LIN {X 0,Y 360.416,Z 365.132,A -85,B 0,C 180,E1 -13245.841,E2 -13245.841} C_VEL
LIN {X 0,Y 360.571,Z 364.155,A -85,B 0,C 180,E1 -13247.25,E2 -13247.25} C_VEL
LIN {X 0,Y 360.971,Z 361.249,A -85,B 0,C 180,E1 -13249.327,E2 -13249.327} C_VEL
LIN {X 0,Y 361.318,Z 358.82,A -85,B 0,C 180,E1 -13250.493,E2 -13250.493} C_VEL
LIN {X 0,Y 361.66,Z 355.683,A -85,B 0,C 180,E1 -13251.666,E2 -13251.666} C_VEL
LIN {X 0,Y 362.259,Z 350.688,A -85,B 0,C 180,E1 -13253.131,E2 -13253.131} C_VEL
LIN {X 0,Y 362.957,Z 344.77,A -85,B 0,C 180,E1 -13254.493,E2 -13254.493} C_VEL
LIN {X 0,Y 363.512,Z 339.656,A -85,B 0,C 180,E1 -13255.477,E2 -13255.477} C_VEL
LIN {X 0,Y 364.34,Z 332.196,A -85,B 0,C 180,E1 -13256.645,E2 -13256.645} C_VEL
LIN {X 0,Y 365.036,Z 325.448,A -85,B 0,C 180,E1 -13257.519,E2 -13257.519} C_VEL
LIN {X 0,Y 365.771,Z 317.345,A -85,B 0,C 180,E1 -13258.378,E2 -13258.378} C_VEL
LIN {X 0,Y 366.188,Z 311.806,A -85,B 0,C 180,E1 -13258.881,E2 -13258.881} C_VEL
LIN {X 0,Y 364.576,Z 302,A -85,B 0,C 180,E1 -13259.701,E2 -13259.701} C_VEL
LIN {X 0,Y 362.216,Z 292.488,A -85,B 0,C 180,E1 -13260.364,E2 -13260.364} C_VEL
LIN {X 0,Y 360.856,Z 287.319,A -85,B 0,C 180,E1 -13260.684,E2 -13260.684} C_VEL
LIN {X 0,Y 360.947,Z 284.654,A -85,B 0,C 180,E1 -13263.154,E2 -13263.154} C_VEL
LIN {X 0,Y 361.044,Z 281.193,A -85,B 0,C 180,E1 -13266.457,E2 -13266.457} C_VEL
LIN {X 0,Y 360.464,Z 280.32,A -85,B 0,C 180,E1 -13267.379,E2 -13267.379} C_VEL
LIN {X 0,Y 357.716,Z 279.131,A -85,B 0,C 180,E1 -13268.886,E2 -13268.886} C_VEL
LIN {X 0,Y 355.368,Z 278.213,A -85,B 0,C 180,E1 -13270.107,E2 -13270.107} C_VEL
LIN {X 0,Y 354.387,Z 277.418,A -85,B 0,C 180,E1 -13271.047,E2 -13271.047} C_VEL
LIN {X 0,Y 354.324,Z 277.117,A -85,B 0,C 180,E1 -13271.364,E2 -13271.364} C_VEL
LIN {X 0,Y 354.508,Z 274.121,A -85,B 0,C 180,E1 -13274.468,E2 -13274.468} C_VEL
LIN {X 0,Y 354.541,Z 273.133,A -85,B 0,C 180,E1 -13275.528,E2 -13275.528} C_VEL
LIN {X 0,Y 354.741,Z 273.111,A -85,B 0,C 180,E1 -13278.834,E2 -13278.834} C_VEL
LIN {X 0,Y 354.791,Z 273.106,A -85,B 0,C 180,E1 -13282.119,E2 -13282.119} C_VEL
LIN {X 0,Y 354.793,Z 273.105,A -85,B 0,C 180,E1 -13284.942,E2 -13284.942} C_VEL
LIN {X 0,Y 354.774,Z 273.106,A -85,B 0,C 180,E1 -13288.407,E2 -13288.407} C_VEL
LIN {X 0,Y 354.828,Z 273.097,A -85,B 0,C 180,E1 -13291.62,E2 -13291.62} C_VEL
LIN {X 0,Y 354.881,Z 273.093,A -85,B 0,C 180,E1 -13294.174,E2 -13294.174} C_VEL
LIN {X 0,Y 354.81,Z 273.101,A -85,B 0,C 180,E1 -13297.895,E2 -13297.895} C_VEL
LIN {X 0,Y 354.907,Z 273.086,A -85,B 0,C 180,E1 -13301.893,E2 -13301.893} C_VEL
LIN {X 0,Y 354.929,Z 273.082,A -85,B 0,C 180,E1 -13305.983,E2 -13305.983} C_VEL
LIN {X 0,Y 354.969,Z 273.078,A -85,B 0,C 180,E1 -13309.738,E2 -13309.738} C_VEL
LIN {X 0,Y 355.087,Z 273.062,A -85,B 0,C 180,E1 -13313.182,E2 -13313.182} C_VEL
LIN {X 0,Y 355.235,Z 273.044,A -85,B 0,C 180,E1 -13317.734,E2 -13317.734} C_VEL
LIN {X 0,Y 355.386,Z 273.029,A -85,B 0,C 180,E1 -13320.002,E2 -13320.002} C_VEL
LIN {X 0,Y 355.232,Z 273.045,A -85,B 0,C 180,E1 -13322.27,E2 -13322.27} C_VEL
LIN {X 0,Y 355.129,Z 273.058,A -85,B 0,C 180,E1 -13326.821,E2 -13326.821} C_VEL
LIN {X 0,Y 355.006,Z 273.076,A -85,B 0,C 180,E1 -13329.114,E2 -13329.114} C_VEL
LIN {X 0,Y 354.916,Z 273.087,A -85,B 0,C 180,E1 -13332.583,E2 -13332.583} C_VEL
LIN {X 0,Y 354.882,Z 273.093,A -85,B 0,C 180,E1 -13336.098,E2 -13336.098} C_VEL
LIN {X 0,Y 354.895,Z 273.091,A -85,B 0,C 180,E1 -13338.474,E2 -13338.474} C_VEL
LIN {X 0,Y 354.808,Z 273.1,A -85,B 0,C 180,E1 -13342.109,E2 -13342.109} C_VEL
LIN {X 0,Y 354.82,Z 273.103,A -85,B 0,C 180,E1 -13345.835,E2 -13345.835} C_VEL
LIN {X 0,Y 354.793,Z 273.107,A -85,B 0,C 180,E1 -13349.686,E2 -13349.686} C_VEL
LIN {X 0,Y 354.781,Z 273.111,A -85,B 0,C 180,E1 -13352.336,E2 -13352.336} C_VEL
LIN {X 0,Y 354.817,Z 273.106,A -85,B 0,C 180,E1 -13355.701,E2 -13355.701} C_VEL
LIN {X 0,Y 354.82,Z 273.101,A -85,B 0,C 180,E1 -13359.426,E2 -13359.426} C_VEL
LIN {X 0,Y 354.801,Z 273.104,A -85,B 0,C 180,E1 -13362.872,E2 -13362.872} C_VEL
LIN {X 0,Y 354.763,Z 273.105,A -85,B 0,C 180,E1 -13366.106,E2 -13366.106} C_VEL
LIN {X 0,Y 354.82,Z 273.147,A -85,B 0,C 180,E1 -13367.669,E2 -13367.669} C_VEL
LIN {X 0,Y 355.607,Z 277.448,A -85,B 0,C 180,E1 -13370.773,E2 -13370.773} C_VEL
LIN {X 0,Y 356.383,Z 282.197,A -85,B 0,C 180,E1 -13373.955,E2 -13373.955} C_VEL
LIN {X 0,Y 356.829,Z 286.286,A -85,B 0,C 180,E1 -13376.534,E2 -13376.534} C_VEL
LIN {X 0,Y 356.512,Z 289.72,A -85,B 0,C 180,E1 -13378.545,E2 -13378.545} C_VEL
LIN {X 0,Y 355.735,Z 295.338,A -85,B 0,C 180,E1 -13381.698,E2 -13381.698} C_VEL
LIN {X 0,Y 354.922,Z 302.58,A -85,B 0,C 180,E1 -13385.628,E2 -13385.628} C_VEL
LIN {X 0,Y 354.219,Z 310.283,A -85,B 0,C 180,E1 -13389.685,E2 -13389.685} C_VEL
LIN {X 0,Y 353.865,Z 316.532,A -85,B 0,C 180,E1 -13392.893,E2 -13392.893} C_VEL
LIN {X 0,Y 356.246,Z 330.063,A -85,B 0,C 180,E1 -13393.674,E2 -13393.674} C_VEL
LIN {X 0,Y 357.341,Z 339.073,A -85,B 0,C 180,E1 -13394.341,E2 -13394.341} C_VEL
LIN {X 0,Y 357.782,Z 346.729,A -85,B 0,C 180,E1 -13395.013,E2 -13395.013} C_VEL
LIN {X 0,Y 357.533,Z 354.246,A -85,B 0,C 180,E1 -13395.778,E2 -13395.778} C_VEL
LIN {X 0,Y 356.617,Z 362.305,A -85,B 0,C 180,E1 -13396.758,E2 -13396.758} C_VEL
LIN {X 0,Y 355.84,Z 368.979,A -85,B 0,C 180,E1 -13397.743,E2 -13397.743} C_VEL
LIN {X 0,Y 355.12,Z 375.328,A -85,B 0,C 180,E1 -13398.876,E2 -13398.876} C_VEL
LIN {X 0,Y 354.531,Z 380.62,A -85,B 0,C 180,E1 -13400.013,E2 -13400.013} C_VEL
LIN {X 0,Y 353.96,Z 386.01,A -85,B 0,C 180,E1 -13401.438,E2 -13401.438} C_VEL
LIN {X 0,Y 353.643,Z 389.518,A -85,B 0,C 180,E1 -13402.58,E2 -13402.58} C_VEL
LIN {X 0,Y 353.349,Z 393.573,A -85,B 0,C 180,E1 -13404.294,E2 -13404.294} C_VEL
LIN {X 0,Y 353.337,Z 395.563,A -85,B 0,C 180,E1 -13405.438,E2 -13405.438} C_VEL
LIN {X 0,Y 353.267,Z 397.05,A -85,B 0,C 180,E1 -13406.58,E2 -13406.58} C_VEL
LIN {X 0,Y 353.258,Z 398.025,A -85,B 0,C 180,E1 -13407.721,E2 -13407.721} C_VEL
LIN {X 0,Y 353.357,Z 398.412,A -85,B 0,C 180,E1 -13408.862,E2 -13408.862} C_VEL
LIN {X 0,Y 353.398,Z 398.321,A -85,B 0,C 180,E1 -13410.001,E2 -13410.001} C_VEL
LIN {X 0,Y 353.396,Z 397.764,A -85,B 0,C 180,E1 -13411.141,E2 -13411.141} C_VEL
LIN {X 0,Y 353.307,Z 396.724,A -85,B 0,C 180,E1 -13412.282,E2 -13412.282} C_VEL
LIN {X 0,Y 353.343,Z 394.041,A -85,B 0,C 180,E1 -13413.993,E2 -13413.993} C_VEL
LIN {X 0,Y 353.358,Z 391.614,A -85,B 0,C 180,E1 -13415.136,E2 -13415.136} C_VEL
LIN {X 0,Y 353.53,Z 386.65,A -85,B 0,C 180,E1 -13416.852,E2 -13416.852} C_VEL
LIN {X 0,Y 353.733,Z 382.491,A -85,B 0,C 180,E1 -13417.996,E2 -13417.996} C_VEL
LIN {X 0,Y 354.012,Z 377.481,A -85,B 0,C 180,E1 -13419.14,E2 -13419.14} C_VEL
LIN {X 0,Y 354.39,Z 371.438,A -85,B 0,C 180,E1 -13420.283,E2 -13420.283} C_VEL
LIN {X 0,Y 354.914,Z 364.082,A -85,B 0,C 180,E1 -13421.423,E2 -13421.423} C_VEL
LIN {X 0,Y 355.487,Z 356.211,A -85,B 0,C 180,E1 -13422.417,E2 -13422.417} C_VEL
LIN {X 0,Y 355.957,Z 349.415,A -85,B 0,C 180,E1 -13423.125,E2 -13423.125} C_VEL
LIN {X 0,Y 355.74,Z 342.879,A -85,B 0,C 180,E1 -13423.715,E2 -13423.715} C_VEL
LIN {X 0,Y 354.992,Z 332.661,A -85,B 0,C 180,E1 -13424.45,E2 -13424.45} C_VEL
LIN {X 0,Y 354.116,Z 322.965,A -85,B 0,C 180,E1 -13424.972,E2 -13424.972} C_VEL
LIN {X 0,Y 353.55,Z 317.049,A -85,B 0,C 180,E1 -13425.236,E2 -13425.236} C_VEL
LIN {X 0,Y 353.827,Z 310.396,A -85,B 0,C 180,E1 -13428.532,E2 -13428.532} C_VEL
LIN {X 0,Y 354.261,Z 303.169,A -85,B 0,C 180,E1 -13432.145,E2 -13432.145} C_VEL
LIN {X 0,Y 354.802,Z 295.919,A -85,B 0,C 180,E1 -13435.836,E2 -13435.836} C_VEL
LIN {X 0,Y 355.492,Z 288.772,A -85,B 0,C 180,E1 -13439.554,E2 -13439.554} C_VEL
LIN {X 0,Y 356.216,Z 282.582,A -85,B 0,C 180,E1 -13442.86,E2 -13442.86} C_VEL
LIN {X 0,Y 355.899,Z 278.88,A -85,B 0,C 180,E1 -13444.938,E2 -13444.938} C_VEL
LIN {X 0,Y 354.887,Z 273.094,A -85,B 0,C 180,E1 -13448.415,E2 -13448.415} C_VEL
LIN {X 0,Y 354.804,Z 273.102,A -85,B 0,C 180,E1 -13452.337,E2 -13452.337} C_VEL
LIN {X 0,Y 354.777,Z 273.107,A -85,B 0,C 180,E1 -13456.103,E2 -13456.103} C_VEL
LIN {X 0,Y 354.797,Z 273.101,A -85,B 0,C 180,E1 -13459.179,E2 -13459.179} C_VEL
LIN {X 0,Y 354.816,Z 273.098,A -85,B 0,C 180,E1 -13462.403,E2 -13462.403} C_VEL
LIN {X 0,Y 354.822,Z 273.098,A -85,B 0,C 180,E1 -13464.94,E2 -13464.94} C_VEL
LIN {X 0,Y 354.803,Z 273.1,A -85,B 0,C 180,E1 -13468.405,E2 -13468.405} C_VEL
LIN {X 0,Y 354.861,Z 273.096,A -85,B 0,C 180,E1 -13471.618,E2 -13471.618} C_VEL
LIN {X 0,Y 354.909,Z 273.087,A -85,B 0,C 180,E1 -13474.172,E2 -13474.172} C_VEL
LIN {X 0,Y 354.827,Z 273.097,A -85,B 0,C 180,E1 -13477.892,E2 -13477.892} C_VEL
LIN {X 0,Y 354.899,Z 273.088,A -85,B 0,C 180,E1 -13481.907,E2 -13481.907} C_VEL
LIN {X 0,Y 354.952,Z 273.081,A -85,B 0,C 180,E1 -13485.98,E2 -13485.98} C_VEL
LIN {X 0,Y 354.964,Z 273.08,A -85,B 0,C 180,E1 -13489.734,E2 -13489.734} C_VEL
LIN {X 0,Y 355.119,Z 273.063,A -85,B 0,C 180,E1 -13493.179,E2 -13493.179} C_VEL
LIN {X 0,Y 355.25,Z 273.044,A -85,B 0,C 180,E1 -13497.73,E2 -13497.73} C_VEL
LIN {X 0,Y 355.381,Z 273.028,A -85,B 0,C 180,E1 -13499.998,E2 -13499.998} C_VEL
LIN {X 0,Y 355.252,Z 273.047,A -85,B 0,C 180,E1 -13502.265,E2 -13502.265} C_VEL
LIN {X 0,Y 355.143,Z 273.059,A -85,B 0,C 180,E1 -13506.817,E2 -13506.817} C_VEL
LIN {X 0,Y 355.02,Z 273.073,A -85,B 0,C 180,E1 -13509.11,E2 -13509.11} C_VEL
LIN {X 0,Y 354.925,Z 273.087,A -85,B 0,C 180,E1 -13512.578,E2 -13512.578} C_VEL
LIN {X 0,Y 354.892,Z 273.093,A -85,B 0,C 180,E1 -13516.093,E2 -13516.093} C_VEL
LIN {X 0,Y 354.905,Z 273.089,A -85,B 0,C 180,E1 -13518.469,E2 -13518.469} C_VEL
LIN {X 0,Y 354.835,Z 273.1,A -85,B 0,C 180,E1 -13522.103,E2 -13522.103} C_VEL
LIN {X 0,Y 354.898,Z 273.092,A -85,B 0,C 180,E1 -13525.825,E2 -13525.825} C_VEL
LIN {X 0,Y 354.815,Z 273.103,A -85,B 0,C 180,E1 -13529.679,E2 -13529.679} C_VEL
LIN {X 0,Y 354.803,Z 273.104,A -85,B 0,C 180,E1 -13533.699,E2 -13533.699} C_VEL
LIN {X 0,Y 354.797,Z 273.1,A -85,B 0,C 180,E1 -13536.456,E2 -13536.456} C_VEL
LIN {X 0,Y 354.818,Z 273.103,A -85,B 0,C 180,E1 -13539.421,E2 -13539.421} C_VEL
LIN {X 0,Y 354.835,Z 273.097,A -85,B 0,C 180,E1 -13542.874,E2 -13542.874} C_VEL
LIN {X 0,Y 354.858,Z 273.093,A -85,B 0,C 180,E1 -13546.116,E2 -13546.116} C_VEL
LIN {X 0,Y 354.847,Z 273.099,A -85,B 0,C 180,E1 -13549.186,E2 -13549.186} C_VEL
LIN {X 0,Y 354.799,Z 273.1,A -85,B 0,C 180,E1 -13552.399,E2 -13552.399} C_VEL
LIN {X 0,Y 354.802,Z 273.105,A -85,B 0,C 180,E1 -13554.938,E2 -13554.938} C_VEL
LIN {X 0,Y 354.781,Z 273.104,A -85,B 0,C 180,E1 -13558.402,E2 -13558.402} C_VEL
LIN {X 0,Y 354.841,Z 273.095,A -85,B 0,C 180,E1 -13561.617,E2 -13561.617} C_VEL
LIN {X 0,Y 354.886,Z 273.09,A -85,B 0,C 180,E1 -13564.17,E2 -13564.17} C_VEL
LIN {X 0,Y 354.835,Z 273.096,A -85,B 0,C 180,E1 -13567.893,E2 -13567.893} C_VEL
LIN {X 0,Y 354.771,Z 273.107,A -85,B 0,C 180,E1 -13570.318,E2 -13570.318} C_VEL
LIN {X 0,Y 354.639,Z 273.124,A -85,B 0,C 180,E1 -13572.705,E2 -13572.705} C_VEL
LIN {X 0,Y 354.215,Z 273.284,A -85,B 0,C 180,E1 -13576.447,E2 -13576.447} C_VEL
LIN {X 0,Y 354.012,Z 276.801,A -85,B 0,C 180,E1 -13579.706,E2 -13579.706} C_VEL
LIN {X 0,Y 354.09,Z 280.552,A -85,B 0,C 180,E1 -13583.159,E2 -13583.159} C_VEL
LIN {X 0,Y 353.926,Z 284.439,A -85,B 0,C 180,E1 -13586.583,E2 -13586.583} C_VEL
LIN {X 0,Y 353.759,Z 287.132,A -85,B 0,C 180,E1 -13588.931,E2 -13588.931} C_VEL
LIN {X 0,Y 355.467,Z 298.103,A -85,B 0,C 180,E1 -13589.503,E2 -13589.503} C_VEL
LIN {X 0,Y 356.869,Z 307.131,A -85,B 0,C 180,E1 -13590.14,E2 -13590.14} C_VEL
LIN {X 0,Y 356.601,Z 315.616,A -85,B 0,C 180,E1 -13590.845,E2 -13590.845} C_VEL
LIN {X 0,Y 356.062,Z 323.845,A -85,B 0,C 180,E1 -13591.695,E2 -13591.695} C_VEL
LIN {X 0,Y 355.513,Z 331.648,A -85,B 0,C 180,E1 -13592.69,E2 -13592.69} C_VEL
LIN {X 0,Y 355.093,Z 338.077,A -85,B 0,C 180,E1 -13593.687,E2 -13593.687} C_VEL
LIN {X 0,Y 354.526,Z 345.642,A -85,B 0,C 180,E1 -13595.116,E2 -13595.116} C_VEL
LIN {X 0,Y 354.214,Z 351.587,A -85,B 0,C 180,E1 -13596.549,E2 -13596.549} C_VEL
LIN {X 0,Y 353.827,Z 356.276,A -85,B 0,C 180,E1 -13597.991,E2 -13597.991} C_VEL
LIN {X 0,Y 353.593,Z 359.314,A -85,B 0,C 180,E1 -13599.148,E2 -13599.148} C_VEL
LIN {X 0,Y 353.412,Z 361.677,A -85,B 0,C 180,E1 -13600.308,E2 -13600.308} C_VEL
LIN {X 0,Y 353.348,Z 363.44,A -85,B 0,C 180,E1 -13601.471,E2 -13601.471} C_VEL
LIN {X 0,Y 353.272,Z 364.919,A -85,B 0,C 180,E1 -13602.903,E2 -13602.903} C_VEL
LIN {X 0,Y 353.249,Z 365.717,A -85,B 0,C 180,E1 -13604.988,E2 -13604.988} C_VEL
LIN {X 0,Y 353.362,Z 365.406,A -85,B 0,C 180,E1 -13606.166,E2 -13606.166} C_VEL
LIN {X 0,Y 353.516,Z 364.468,A -85,B 0,C 180,E1 -13607.408,E2 -13607.408} C_VEL
LIN {X 0,Y 353.722,Z 363.108,A -85,B 0,C 180,E1 -13608.534,E2 -13608.534} C_VEL
LIN {X 0,Y 354.198,Z 359.965,A -85,B 0,C 180,E1 -13610.316,E2 -13610.316} C_VEL
LIN {X 0,Y 354.757,Z 355.346,A -85,B 0,C 180,E1 -13612.109,E2 -13612.109} C_VEL
LIN {X 0,Y 355.445,Z 350.134,A -85,B 0,C 180,E1 -13613.601,E2 -13613.601} C_VEL
LIN {X 0,Y 356.082,Z 345.008,A -85,B 0,C 180,E1 -13614.79,E2 -13614.79} C_VEL
LIN {X 0,Y 356.705,Z 338.68,A -85,B 0,C 180,E1 -13615.999,E2 -13615.999} C_VEL
LIN {X 0,Y 357.586,Z 332.042,A -85,B 0,C 180,E1 -13617.031,E2 -13617.031} C_VEL
LIN {X 0,Y 358.34,Z 325.174,A -85,B 0,C 180,E1 -13617.922,E2 -13617.922} C_VEL
LIN {X 0,Y 359.065,Z 317.277,A -85,B 0,C 180,E1 -13618.765,E2 -13618.765} C_VEL
LIN {X 0,Y 359.325,Z 311.85,A -85,B 0,C 180,E1 -13619.271,E2 -13619.271} C_VEL
LIN {X 0,Y 357.496,Z 301.944,A -85,B 0,C 180,E1 -13620.124,E2 -13620.124} C_VEL
LIN {X 0,Y 355.149,Z 292.733,A -85,B 0,C 180,E1 -13620.784,E2 -13620.784} C_VEL
LIN {X 0,Y 353.805,Z 287.658,A -85,B 0,C 180,E1 -13621.126,E2 -13621.126} C_VEL
LIN {X 0,Y 353.887,Z 284.831,A -85,B 0,C 180,E1 -13623.782,E2 -13623.782} C_VEL
LIN {X 0,Y 354.094,Z 280.511,A -85,B 0,C 180,E1 -13627.97,E2 -13627.97} C_VEL
LIN {X 0,Y 354.324,Z 277.117,A -85,B 0,C 180,E1 -13631.364,E2 -13631.364} C_VEL
LIN {X 0,Y 353.706,Z 276.302,A -85,B 0,C 180,E1 -13632.304,E2 -13632.304} C_VEL
LIN {X 0,Y 350.908,Z 275.228,A -85,B 0,C 180,E1 -13633.84,E2 -13633.84} C_VEL
LIN {X 0,Y 348.554,Z 274.602,A -85,B 0,C 180,E1 -13635.088,E2 -13635.088} C_VEL
LIN {X 0,Y 347.597,Z 274.201,A -85,B 0,C 180,E1 -13636.053,E2 -13636.053} C_VEL
LIN {X 0,Y 347.549,Z 274.075,A -85,B 0,C 180,E1 -13636.38,E2 -13636.38} C_VEL
LIN {X 0,Y 347.699,Z 273.989,A -85,B 0,C 180,E1 -13639.702,E2 -13639.702} C_VEL
LIN {X 0,Y 347.747,Z 273.986,A -85,B 0,C 180,E1 -13642.681,E2 -13642.681} C_VEL
LIN {X 0,Y 347.729,Z 273.985,A -85,B 0,C 180,E1 -13645.957,E2 -13645.957} C_VEL
LIN {X 0,Y 347.731,Z 273.983,A -85,B 0,C 180,E1 -13649.653,E2 -13649.653} C_VEL
LIN {X 0,Y 347.813,Z 273.973,A -85,B 0,C 180,E1 -13653.609,E2 -13653.609} C_VEL
LIN {X 0,Y 347.769,Z 273.975,A -85,B 0,C 180,E1 -13656.163,E2 -13656.163} C_VEL
LIN {X 0,Y 347.795,Z 273.974,A -85,B 0,C 180,E1 -13659.911,E2 -13659.911} C_VEL
LIN {X 0,Y 347.851,Z 273.964,A -85,B 0,C 180,E1 -13662.361,E2 -13662.361} C_VEL
LIN {X 0,Y 347.883,Z 273.96,A -85,B 0,C 180,E1 -13665.973,E2 -13665.973} C_VEL
LIN {X 0,Y 347.919,Z 273.956,A -85,B 0,C 180,E1 -13669.528,E2 -13669.528} C_VEL
LIN {X 0,Y 348.055,Z 273.939,A -85,B 0,C 180,E1 -13673.044,E2 -13673.044} C_VEL
LIN {X 0,Y 348.198,Z 273.92,A -85,B 0,C 180,E1 -13677.689,E2 -13677.689} C_VEL
LIN {X 0,Y 348.334,Z 273.907,A -85,B 0,C 180,E1 -13680.002,E2 -13680.002} C_VEL
LIN {X 0,Y 348.195,Z 273.922,A -85,B 0,C 180,E1 -13682.316,E2 -13682.316} C_VEL
LIN {X 0,Y 348.097,Z 273.935,A -85,B 0,C 180,E1 -13686.96,E2 -13686.96} C_VEL
LIN {X 0,Y 347.959,Z 273.954,A -85,B 0,C 180,E1 -13689.301,E2 -13689.301} C_VEL
LIN {X 0,Y 347.884,Z 273.964,A -85,B 0,C 180,E1 -13692.842,E2 -13692.842} C_VEL
LIN {X 0,Y 347.831,Z 273.972,A -85,B 0,C 180,E1 -13696.434,E2 -13696.434} C_VEL
LIN {X 0,Y 347.844,Z 273.968,A -85,B 0,C 180,E1 -13698.863,E2 -13698.863} C_VEL
LIN {X 0,Y 347.752,Z 273.981,A -85,B 0,C 180,E1 -13702.583,E2 -13702.583} C_VEL
LIN {X 0,Y 347.769,Z 273.979,A -85,B 0,C 180,E1 -13705.114,E2 -13705.114} C_VEL
LIN {X 0,Y 347.735,Z 273.988,A -85,B 0,C 180,E1 -13707.702,E2 -13707.702} C_VEL
LIN {X 0,Y 347.735,Z 273.987,A -85,B 0,C 180,E1 -13710.351,E2 -13710.351} C_VEL
LIN {X 0,Y 347.743,Z 273.987,A -85,B 0,C 180,E1 -13714.046,E2 -13714.046} C_VEL
LIN {X 0,Y 347.758,Z 273.983,A -85,B 0,C 180,E1 -13717.323,E2 -13717.323} C_VEL
LIN {X 0,Y 347.752,Z 273.983,A -85,B 0,C 180,E1 -13720.296,E2 -13720.296} C_VEL
LIN {X 0,Y 347.741,Z 273.986,A -85,B 0,C 180,E1 -13723.407,E2 -13723.407} C_VEL
LIN {X 0,Y 347.758,Z 274.009,A -85,B 0,C 180,E1 -13727.195,E2 -13727.195} C_VEL
LIN {X 0,Y 348.479,Z 277.803,A -85,B 0,C 180,E1 -13730.031,E2 -13730.031} C_VEL
LIN {X 0,Y 349.3,Z 282.923,A -85,B 0,C 180,E1 -13733.594,E2 -13733.594} C_VEL
LIN {X 0,Y 349.785,Z 286.252,A -85,B 0,C 180,E1 -13735.767,E2 -13735.767} C_VEL
LIN {X 0,Y 349.706,Z 289.194,A -85,B 0,C 180,E1 -13737.574,E2 -13737.574} C_VEL
LIN {X 0,Y 348.863,Z 295.253,A -85,B 0,C 180,E1 -13741.088,E2 -13741.088} C_VEL
LIN {X 0,Y 347.928,Z 302.918,A -85,B 0,C 180,E1 -13745.367,E2 -13745.367} C_VEL
LIN {X 0,Y 347.212,Z 310.139,A -85,B 0,C 180,E1 -13749.256,E2 -13749.256} C_VEL
LIN {X 0,Y 346.862,Z 316.196,A -85,B 0,C 180,E1 -13752.46,E2 -13752.46} C_VEL
LIN {X 0,Y 349.142,Z 328.662,A -85,B 0,C 180,E1 -13753.182,E2 -13753.182} C_VEL
LIN {X 0,Y 350.371,Z 338.461,A -85,B 0,C 180,E1 -13753.92,E2 -13753.92} C_VEL
LIN {X 0,Y 350.919,Z 347.311,A -85,B 0,C 180,E1 -13754.727,E2 -13754.727} C_VEL
LIN {X 0,Y 350.678,Z 354.545,A -85,B 0,C 180,E1 -13755.494,E2 -13755.494} C_VEL
LIN {X 0,Y 349.733,Z 362.497,A -85,B 0,C 180,E1 -13756.492,E2 -13756.492} C_VEL
LIN {X 0,Y 348.911,Z 369.085,A -85,B 0,C 180,E1 -13757.496,E2 -13757.496} C_VEL
LIN {X 0,Y 348.147,Z 375.36,A -85,B 0,C 180,E1 -13758.65,E2 -13758.65} C_VEL
LIN {X 0,Y 347.519,Z 380.589,A -85,B 0,C 180,E1 -13759.809,E2 -13759.809} C_VEL
LIN {X 0,Y 346.918,Z 385.924,A -85,B 0,C 180,E1 -13761.262,E2 -13761.262} C_VEL
LIN {X 0,Y 346.572,Z 389.38,A -85,B 0,C 180,E1 -13762.427,E2 -13762.427} C_VEL
LIN {X 0,Y 346.273,Z 393.387,A -85,B 0,C 180,E1 -13764.177,E2 -13764.177} C_VEL
LIN {X 0,Y 346.25,Z 395.333,A -85,B 0,C 180,E1 -13765.345,E2 -13765.345} C_VEL
LIN {X 0,Y 346.19,Z 396.779,A -85,B 0,C 180,E1 -13766.51,E2 -13766.51} C_VEL
LIN {X 0,Y 346.164,Z 397.734,A -85,B 0,C 180,E1 -13767.674,E2 -13767.674} C_VEL
LIN {X 0,Y 346.258,Z 398.101,A -85,B 0,C 180,E1 -13768.839,E2 -13768.839} C_VEL
LIN {X 0,Y 346.319,Z 397.971,A -85,B 0,C 180,E1 -13770.002,E2 -13770.002} C_VEL
LIN {X 0,Y 346.3,Z 397.374,A -85,B 0,C 180,E1 -13771.164,E2 -13771.164} C_VEL
LIN {X 0,Y 346.212,Z 396.296,A -85,B 0,C 180,E1 -13772.328,E2 -13772.328} C_VEL
LIN {X 0,Y 346.274,Z 393.57,A -85,B 0,C 180,E1 -13774.075,E2 -13774.075} C_VEL
LIN {X 0,Y 346.294,Z 389.563,A -85,B 0,C 180,E1 -13775.826,E2 -13775.826} C_VEL
LIN {X 0,Y 346.456,Z 386.081,A -85,B 0,C 180,E1 -13776.992,E2 -13776.992} C_VEL
LIN {X 0,Y 346.742,Z 380.681,A -85,B 0,C 180,E1 -13778.452,E2 -13778.452} C_VEL
LIN {X 0,Y 347.145,Z 373.928,A -85,B 0,C 180,E1 -13779.91,E2 -13779.91} C_VEL
LIN {X 0,Y 347.75,Z 365.286,A -85,B 0,C 180,E1 -13781.366,E2 -13781.366} C_VEL
LIN {X 0,Y 348.312,Z 357.723,A -85,B 0,C 180,E1 -13782.381,E2 -13782.381} C_VEL
LIN {X 0,Y 348.921,Z 349.822,A -85,B 0,C 180,E1 -13783.246,E2 -13783.246} C_VEL
LIN {X 0,Y 348.599,Z 341.532,A -85,B 0,C 180,E1 -13784.002,E2 -13784.002} C_VEL
LIN {X 0,Y 348.004,Z 333.338,A -85,B 0,C 180,E1 -13784.607,E2 -13784.607} C_VEL
LIN {X 0,Y 347.135,Z 323.58,A -85,B 0,C 180,E1 -13785.159,E2 -13785.159} C_VEL
LIN {X 0,Y 346.498,Z 316.756,A -85,B 0,C 180,E1 -13785.478,E2 -13785.478} C_VEL
LIN {X 0,Y 346.753,Z 309.946,A -85,B 0,C 180,E1 -13788.924,E2 -13788.924} C_VEL
LIN {X 0,Y 347.236,Z 302.74,A -85,B 0,C 180,E1 -13792.618,E2 -13792.618} C_VEL
LIN {X 0,Y 347.827,Z 295.491,A -85,B 0,C 180,E1 -13796.394,E2 -13796.394} C_VEL
LIN {X 0,Y 348.625,Z 288.264,A -85,B 0,C 180,E1 -13800.265,E2 -13800.265} C_VEL
LIN {X 0,Y 349.192,Z 283.406,A -85,B 0,C 180,E1 -13802.918,E2 -13802.918} C_VEL
LIN {X 0,Y 348.845,Z 279.72,A -85,B 0,C 180,E1 -13805.043,E2 -13805.043} C_VEL
LIN {X 0,Y 347.845,Z 273.971,A -85,B 0,C 180,E1 -13808.57,E2 -13808.57} C_VEL
LIN {X 0,Y 347.76,Z 273.98,A -85,B 0,C 180,E1 -13811.83,E2 -13811.83} C_VEL
LIN {X 0,Y 347.715,Z 273.982,A -85,B 0,C 180,E1 -13815.027,E2 -13815.027} C_VEL
LIN {X 0,Y 347.76,Z 273.978,A -85,B 0,C 180,E1 -13818.397,E2 -13818.397} C_VEL
LIN {X 0,Y 347.782,Z 273.977,A -85,B 0,C 180,E1 -13822.011,E2 -13822.011} C_VEL
LIN {X 0,Y 347.754,Z 273.982,A -85,B 0,C 180,E1 -13825.536,E2 -13825.536} C_VEL
LIN {X 0,Y 347.774,Z 273.979,A -85,B 0,C 180,E1 -13829.653,E2 -13829.653} C_VEL
LIN {X 0,Y 347.862,Z 273.964,A -85,B 0,C 180,E1 -13832.744,E2 -13832.744} C_VEL
LIN {X 0,Y 347.795,Z 273.972,A -85,B 0,C 180,E1 -13836.161,E2 -13836.161} C_VEL
LIN {X 0,Y 347.809,Z 273.971,A -85,B 0,C 180,E1 -13839.907,E2 -13839.907} C_VEL
LIN {X 0,Y 347.841,Z 273.968,A -85,B 0,C 180,E1 -13843.567,E2 -13843.567} C_VEL
LIN {X 0,Y 347.898,Z 273.964,A -85,B 0,C 180,E1 -13847.159,E2 -13847.159} C_VEL
LIN {X 0,Y 347.943,Z 273.958,A -85,B 0,C 180,E1 -13850.699,E2 -13850.699} C_VEL
LIN {X 0,Y 348.085,Z 273.94,A -85,B 0,C 180,E1 -13853.04,E2 -13853.04} C_VEL
LIN {X 0,Y 348.212,Z 273.92,A -85,B 0,C 180,E1 -13857.685,E2 -13857.685} C_VEL
LIN {X 0,Y 348.332,Z 273.906,A -85,B 0,C 180,E1 -13859.998,E2 -13859.998} C_VEL
LIN {X 0,Y 348.214,Z 273.924,A -85,B 0,C 180,E1 -13862.311,E2 -13862.311} C_VEL
LIN {X 0,Y 348.111,Z 273.934,A -85,B 0,C 180,E1 -13866.955,E2 -13866.955} C_VEL
LIN {X 0,Y 347.972,Z 273.95,A -85,B 0,C 180,E1 -13869.296,E2 -13869.296} C_VEL
LIN {X 0,Y 347.893,Z 273.961,A -85,B 0,C 180,E1 -13872.837,E2 -13872.837} C_VEL
LIN {X 0,Y 347.841,Z 273.969,A -85,B 0,C 180,E1 -13876.429,E2 -13876.429} C_VEL
LIN {X 0,Y 347.854,Z 273.965,A -85,B 0,C 180,E1 -13878.858,E2 -13878.858} C_VEL
LIN {X 0,Y 347.774,Z 273.976,A -85,B 0,C 180,E1 -13882.577,E2 -13882.577} C_VEL
LIN {X 0,Y 347.811,Z 273.97,A -85,B 0,C 180,E1 -13885.106,E2 -13885.106} C_VEL
LIN {X 0,Y 347.807,Z 273.976,A -85,B 0,C 180,E1 -13887.691,E2 -13887.691} C_VEL
LIN {X 0,Y 347.747,Z 273.979,A -85,B 0,C 180,E1 -13890.345,E2 -13890.345} C_VEL
LIN {X 0,Y 347.745,Z 273.98,A -85,B 0,C 180,E1 -13894.041,E2 -13894.041} C_VEL
LIN {X 0,Y 347.762,Z 273.98,A -85,B 0,C 180,E1 -13897.317,E2 -13897.317} C_VEL
LIN {X 0,Y 347.788,Z 273.973,A -85,B 0,C 180,E1 -13900.286,E2 -13900.286} C_VEL
LIN {X 0,Y 347.812,Z 273.975,A -85,B 0,C 180,E1 -13903.39,E2 -13903.39} C_VEL
LIN {X 0,Y 347.809,Z 273.972,A -85,B 0,C 180,E1 -13906.667,E2 -13906.667} C_VEL
LIN {X 0,Y 347.777,Z 273.974,A -85,B 0,C 180,E1 -13910.163,E2 -13910.163} C_VEL
LIN {X 0,Y 347.778,Z 273.974,A -85,B 0,C 180,E1 -13914.122,E2 -13914.122} C_VEL
LIN {X 0,Y 347.727,Z 273.981,A -85,B 0,C 180,E1 -13918.083,E2 -13918.083} C_VEL
LIN {X 0,Y 347.794,Z 273.976,A -85,B 0,C 180,E1 -13920.988,E2 -13920.988} C_VEL
LIN {X 0,Y 347.819,Z 273.969,A -85,B 0,C 180,E1 -13923.605,E2 -13923.605} C_VEL
LIN {X 0,Y 347.784,Z 273.975,A -85,B 0,C 180,E1 -13926.16,E2 -13926.16} C_VEL
LIN {X 0,Y 347.831,Z 273.972,A -85,B 0,C 180,E1 -13928.671,E2 -13928.671} C_VEL
LIN {X 0,Y 347.649,Z 273.995,A -85,B 0,C 180,E1 -13932.346,E2 -13932.346} C_VEL
LIN {X 0,Y 347.159,Z 274.058,A -85,B 0,C 180,E1 -13936.329,E2 -13936.329} C_VEL
LIN {X 0,Y 346.963,Z 277.282,A -85,B 0,C 180,E1 -13939.495,E2 -13939.495} C_VEL
LIN {X 0,Y 347.053,Z 281.082,A -85,B 0,C 180,E1 -13943.02,E2 -13943.02} C_VEL
LIN {X 0,Y 346.871,Z 284.963,A -85,B 0,C 180,E1 -13946.514,E2 -13946.514} C_VEL
LIN {X 0,Y 346.724,Z 287.409,A -85,B 0,C 180,E1 -13948.692,E2 -13948.692} C_VEL
LIN {X 0,Y 348.385,Z 298.392,A -85,B 0,C 180,E1 -13949.276,E2 -13949.276} C_VEL
LIN {X 0,Y 349.667,Z 306.56,A -85,B 0,C 180,E1 -13949.855,E2 -13949.855} C_VEL
LIN {X 0,Y 349.862,Z 311.963,A -85,B 0,C 180,E1 -13950.286,E2 -13950.286} C_VEL
LIN {X 0,Y 349.167,Z 322.273,A -85,B 0,C 180,E1 -13951.296,E2 -13951.296} C_VEL
LIN {X 0,Y 348.636,Z 330.384,A -85,B 0,C 180,E1 -13952.309,E2 -13952.309} C_VEL
LIN {X 0,Y 348.191,Z 336.236,A -85,B 0,C 180,E1 -13953.18,E2 -13953.18} C_VEL
LIN {X 0,Y 347.744,Z 342.722,A -85,B 0,C 180,E1 -13954.345,E2 -13954.345} C_VEL
LIN {X 0,Y 347.303,Z 348.13,A -85,B 0,C 180,E1 -13955.514,E2 -13955.514} C_VEL
LIN {X 0,Y 347.172,Z 351.629,A -85,B 0,C 180,E1 -13956.391,E2 -13956.391} C_VEL
LIN {X 0,Y 346.712,Z 357.163,A -85,B 0,C 180,E1 -13958.156,E2 -13958.156} C_VEL
LIN {X 0,Y 346.391,Z 361.257,A -85,B 0,C 180,E1 -13959.929,E2 -13959.929} C_VEL
LIN {X 0,Y 346.229,Z 364.075,A -85,B 0,C 180,E1 -13961.71,E2 -13961.71} C_VEL
LIN {X 0,Y 346.182,Z 365.28,A -85,B 0,C 180,E1 -13962.989,E2 -13962.989} C_VEL
LIN {X 0,Y 346.133,Z 365.846,A -85,B 0,C 180,E1 -13964.101,E2 -13964.101} C_VEL
LIN {X 0,Y 346.174,Z 365.993,A -85,B 0,C 180,E1 -13965.301,E2 -13965.301} C_VEL
LIN {X 0,Y 346.329,Z 365.634,A -85,B 0,C 180,E1 -13966.503,E2 -13966.503} C_VEL
LIN {X 0,Y 346.498,Z 364.673,A -85,B 0,C 180,E1 -13967.711,E2 -13967.711} C_VEL
LIN {X 0,Y 346.882,Z 362.229,A -85,B 0,C 180,E1 -13969.528,E2 -13969.528} C_VEL
LIN {X 0,Y 347.25,Z 359.856,A -85,B 0,C 180,E1 -13970.742,E2 -13970.742} C_VEL
LIN {X 0,Y 347.873,Z 354.957,A -85,B 0,C 180,E1 -13972.571,E2 -13972.571} C_VEL
LIN {X 0,Y 348.469,Z 350.794,A -85,B 0,C 180,E1 -13973.787,E2 -13973.787} C_VEL
LIN {X 0,Y 349.239,Z 345.204,A -85,B 0,C 180,E1 -13975.108,E2 -13975.108} C_VEL
LIN {X 0,Y 349.803,Z 339.493,A -85,B 0,C 180,E1 -13976.23,E2 -13976.23} C_VEL
LIN {X 0,Y 350.839,Z 331.886,A -85,B 0,C 180,E1 -13977.433,E2 -13977.433} C_VEL
LIN {X 0,Y 351.603,Z 325.241,A -85,B 0,C 180,E1 -13978.302,E2 -13978.302} C_VEL
LIN {X 0,Y 352.318,Z 317.994,A -85,B 0,C 180,E1 -13979.091,E2 -13979.091} C_VEL
LIN {X 0,Y 352.574,Z 313.191,A -85,B 0,C 180,E1 -13979.559,E2 -13979.559} C_VEL
LIN {X 0,Y 350.689,Z 302.799,A -85,B 0,C 180,E1 -13980.493,E2 -13980.493} C_VEL
LIN {X 0,Y 348.32,Z 293.73,A -85,B 0,C 180,E1 -13981.177,E2 -13981.177} C_VEL
LIN {X 0,Y 346.754,Z 288.006,A -85,B 0,C 180,E1 -13981.571,E2 -13981.571} C_VEL
LIN {X 0,Y 346.854,Z 284.873,A -85,B 0,C 180,E1 -13984.563,E2 -13984.563} C_VEL
LIN {X 0,Y 347.066,Z 281.564,A -85,B 0,C 180,E1 -13987.844,E2 -13987.844} C_VEL
LIN {X 0,Y 347.345,Z 277.583,A -85,B 0,C 180,E1 -13991.888,E2 -13991.888} C_VEL
LIN {X 0,Y 347.497,Z 274.581,A -85,B 0,C 180,E1 -13995.059,E2 -13995.059} C_VEL
LIN {X 0,Y 347.549,Z 274.075,A -85,B 0,C 180,E1 -13996.38,E2 -13996.38} C_VEL
LIN {X 0,Y 347.294,Z 274.035,A -85,B 0,C 180,E1 -13997.027,E2 -13997.027} C_VEL
LIN {X 0,Y 345.416,Z 274.273,A -85,B 0,C 180,E1 -13998.298,E2 -13998.298} C_VEL
LIN {X 0,Y 341.742,Z 274.75,A -85,B 0,C 180,E1 -14000.201,E2 -14000.201} C_VEL
LIN {X 0,Y 340.745,Z 274.857,A -85,B 0,C 180,E1 -14001.19,E2 -14001.19} C_VEL
LIN {X 0,Y 340.686,Z 274.863,A -85,B 0,C 180,E1 -14001.524,E2 -14001.524} C_VEL
LIN {X 0,Y 340.7,Z 274.861,A -85,B 0,C 180,E1 -14004.722,E2 -14004.722} C_VEL
LIN {X 0,Y 340.679,Z 274.862,A -85,B 0,C 180,E1 -14008.957,E2 -14008.957} C_VEL
LIN {X 0,Y 340.786,Z 274.848,A -85,B 0,C 180,E1 -14013.021,E2 -14013.021} C_VEL
LIN {X 0,Y 340.737,Z 274.852,A -85,B 0,C 180,E1 -14015.64,E2 -14015.64} C_VEL
LIN {X 0,Y 340.723,Z 274.853,A -85,B 0,C 180,E1 -14019.475,E2 -14019.475} C_VEL
LIN {X 0,Y 340.843,Z 274.837,A -85,B 0,C 180,E1 -14021.986,E2 -14021.986} C_VEL
LIN {X 0,Y 340.855,Z 274.835,A -85,B 0,C 180,E1 -14025.707,E2 -14025.707} C_VEL
LIN {X 0,Y 340.862,Z 274.836,A -85,B 0,C 180,E1 -14029.308,E2 -14029.308} C_VEL
LIN {X 0,Y 341.003,Z 274.818,A -85,B 0,C 180,E1 -14032.899,E2 -14032.899} C_VEL
LIN {X 0,Y 341.159,Z 274.797,A -85,B 0,C 180,E1 -14037.641,E2 -14037.641} C_VEL
LIN {X 0,Y 341.285,Z 274.785,A -85,B 0,C 180,E1 -14040.002,E2 -14040.002} C_VEL
LIN {X 0,Y 341.157,Z 274.798,A -85,B 0,C 180,E1 -14042.363,E2 -14042.363} C_VEL
LIN {X 0,Y 341.066,Z 274.812,A -85,B 0,C 180,E1 -14047.104,E2 -14047.104} C_VEL
LIN {X 0,Y 340.864,Z 274.838,A -85,B 0,C 180,E1 -14050.696,E2 -14050.696} C_VEL
LIN {X 0,Y 340.855,Z 274.839,A -85,B 0,C 180,E1 -14054.327,E2 -14054.327} C_VEL
LIN {X 0,Y 340.83,Z 274.843,A -85,B 0,C 180,E1 -14058.469,E2 -14058.469} C_VEL
LIN {X 0,Y 340.711,Z 274.857,A -85,B 0,C 180,E1 -14061.844,E2 -14061.844} C_VEL
LIN {X 0,Y 340.745,Z 274.855,A -85,B 0,C 180,E1 -14064.84,E2 -14064.84} C_VEL
LIN {X 0,Y 340.679,Z 274.864,A -85,B 0,C 180,E1 -14068.327,E2 -14068.327} C_VEL
LIN {X 0,Y 340.689,Z 274.866,A -85,B 0,C 180,E1 -14071.047,E2 -14071.047} C_VEL
LIN {X 0,Y 340.713,Z 274.862,A -85,B 0,C 180,E1 -14075.281,E2 -14075.281} C_VEL
LIN {X 0,Y 340.709,Z 274.861,A -85,B 0,C 180,E1 -14078.389,E2 -14078.389} C_VEL
LIN {X 0,Y 340.728,Z 274.858,A -85,B 0,C 180,E1 -14082.054,E2 -14082.054} C_VEL
LIN {X 0,Y 340.65,Z 274.863,A -85,B 0,C 180,E1 -14086.229,E2 -14086.229} C_VEL
LIN {X 0,Y 340.761,Z 275.103,A -85,B 0,C 180,E1 -14086.901,E2 -14086.901} C_VEL
LIN {X 0,Y 341.575,Z 279.656,A -85,B 0,C 180,E1 -14090.372,E2 -14090.372} C_VEL
LIN {X 0,Y 342.49,Z 285.133,A -85,B 0,C 180,E1 -14094.211,E2 -14094.211} C_VEL
LIN {X 0,Y 342.844,Z 288.451,A -85,B 0,C 180,E1 -14096.396,E2 -14096.396} C_VEL
LIN {X 0,Y 342.298,Z 292.935,A -85,B 0,C 180,E1 -14099.119,E2 -14099.119} C_VEL
LIN {X 0,Y 341.556,Z 298.233,A -85,B 0,C 180,E1 -14102.227,E2 -14102.227} C_VEL
LIN {X 0,Y 340.81,Z 304.284,A -85,B 0,C 180,E1 -14105.644,E2 -14105.644} C_VEL
LIN {X 0,Y 340.123,Z 311.146,A -85,B 0,C 180,E1 -14109.437,E2 -14109.437} C_VEL
LIN {X 0,Y 339.818,Z 315.861,A -85,B 0,C 180,E1 -14111.994,E2 -14111.994} C_VEL
LIN {X 0,Y 342.31,Z 329.01,A -85,B 0,C 180,E1 -14112.793,E2 -14112.793} C_VEL
LIN {X 0,Y 343.572,Z 339.249,A -85,B 0,C 180,E1 -14113.601,E2 -14113.601} C_VEL
LIN {X 0,Y 344.068,Z 347.923,A -85,B 0,C 180,E1 -14114.429,E2 -14114.429} C_VEL
LIN {X 0,Y 343.816,Z 354.861,A -85,B 0,C 180,E1 -14115.198,E2 -14115.198} C_VEL
LIN {X 0,Y 342.976,Z 361.68,A -85,B 0,C 180,E1 -14116.07,E2 -14116.07} C_VEL
LIN {X 0,Y 342.188,Z 367.492,A -85,B 0,C 180,E1 -14116.945,E2 -14116.945} C_VEL
LIN {X 0,Y 341.381,Z 373.973,A -85,B 0,C 180,E1 -14118.121,E2 -14118.121} C_VEL
LIN {X 0,Y 340.694,Z 379.383,A -85,B 0,C 180,E1 -14119.302,E2 -14119.302} C_VEL
LIN {X 0,Y 340.112,Z 383.916,A -85,B 0,C 180,E1 -14120.486,E2 -14120.486} C_VEL
LIN {X 0,Y 339.697,Z 387.703,A -85,B 0,C 180,E1 -14121.675,E2 -14121.675} C_VEL
LIN {X 0,Y 339.303,Z 392.039,A -85,B 0,C 180,E1 -14123.461,E2 -14123.461} C_VEL
LIN {X 0,Y 339.148,Z 395.104,A -85,B 0,C 180,E1 -14125.247,E2 -14125.247} C_VEL
LIN {X 0,Y 339.115,Z 396.509,A -85,B 0,C 180,E1 -14126.437,E2 -14126.437} C_VEL
LIN {X 0,Y 339.074,Z 397.436,A -85,B 0,C 180,E1 -14127.626,E2 -14127.626} C_VEL
LIN {X 0,Y 339.16,Z 397.79,A -85,B 0,C 180,E1 -14128.814,E2 -14128.814} C_VEL
LIN {X 0,Y 339.227,Z 397.619,A -85,B 0,C 180,E1 -14130.002,E2 -14130.002} C_VEL
LIN {X 0,Y 339.204,Z 396.981,A -85,B 0,C 180,E1 -14131.189,E2 -14131.189} C_VEL
LIN {X 0,Y 339.119,Z 395.86,A -85,B 0,C 180,E1 -14132.377,E2 -14132.377} C_VEL
LIN {X 0,Y 339.205,Z 393.091,A -85,B 0,C 180,E1 -14134.16,E2 -14134.16} C_VEL
LIN {X 0,Y 339.213,Z 388.879,A -85,B 0,C 180,E1 -14136.008,E2 -14136.008} C_VEL
LIN {X 0,Y 339.521,Z 383.554,A -85,B 0,C 180,E1 -14137.734,E2 -14137.734} C_VEL
LIN {X 0,Y 339.848,Z 377.524,A -85,B 0,C 180,E1 -14139.224,E2 -14139.224} C_VEL
LIN {X 0,Y 340.249,Z 371.619,A -85,B 0,C 180,E1 -14140.414,E2 -14140.414} C_VEL
LIN {X 0,Y 340.76,Z 364.422,A -85,B 0,C 180,E1 -14141.602,E2 -14141.602} C_VEL
LIN {X 0,Y 341.375,Z 356.754,A -85,B 0,C 180,E1 -14142.637,E2 -14142.637} C_VEL
LIN {X 0,Y 341.894,Z 350.221,A -85,B 0,C 180,E1 -14143.372,E2 -14143.372} C_VEL
LIN {X 0,Y 341.582,Z 342.11,A -85,B 0,C 180,E1 -14144.143,E2 -14144.143} C_VEL
LIN {X 0,Y 340.918,Z 332.799,A -85,B 0,C 180,E1 -14144.85,E2 -14144.85} C_VEL
LIN {X 0,Y 340.094,Z 323.408,A -85,B 0,C 180,E1 -14145.393,E2 -14145.393} C_VEL
LIN {X 0,Y 339.422,Z 316.415,A -85,B 0,C 180,E1 -14145.732,E2 -14145.732} C_VEL
LIN {X 0,Y 339.692,Z 309.499,A -85,B 0,C 180,E1 -14149.333,E2 -14149.333} C_VEL
LIN {X 0,Y 340.226,Z 302.301,A -85,B 0,C 180,E1 -14153.11,E2 -14153.11} C_VEL
LIN {X 0,Y 340.852,Z 295.096,A -85,B 0,C 180,E1 -14156.977,E2 -14156.977} C_VEL
LIN {X 0,Y 341.694,Z 287.862,A -85,B 0,C 180,E1 -14160.946,E2 -14160.946} C_VEL
LIN {X 0,Y 342.063,Z 284.886,A -85,B 0,C 180,E1 -14162.605,E2 -14162.605} C_VEL
LIN {X 0,Y 341.909,Z 281.32,A -85,B 0,C 180,E1 -14164.692,E2 -14164.692} C_VEL
LIN {X 0,Y 340.891,Z 275.283,A -85,B 0,C 180,E1 -14168.423,E2 -14168.423} C_VEL
LIN {X 0,Y 340.774,Z 274.85,A -85,B 0,C 180,E1 -14168.764,E2 -14168.764} C_VEL
LIN {X 0,Y 340.686,Z 274.858,A -85,B 0,C 180,E1 -14172.904,E2 -14172.904} C_VEL
LIN {X 0,Y 340.686,Z 274.858,A -85,B 0,C 180,E1 -14177.095,E2 -14177.095} C_VEL
LIN {X 0,Y 340.709,Z 274.856,A -85,B 0,C 180,E1 -14180.247,E2 -14180.247} C_VEL
LIN {X 0,Y 340.72,Z 274.858,A -85,B 0,C 180,E1 -14183.559,E2 -14183.559} C_VEL
LIN {X 0,Y 340.702,Z 274.857,A -85,B 0,C 180,E1 -14186.153,E2 -14186.153} C_VEL
LIN {X 0,Y 340.785,Z 274.845,A -85,B 0,C 180,E1 -14190.332,E2 -14190.332} C_VEL
LIN {X 0,Y 340.815,Z 274.844,A -85,B 0,C 180,E1 -14193.019,E2 -14193.019} C_VEL
LIN {X 0,Y 340.765,Z 274.851,A -85,B 0,C 180,E1 -14195.637,E2 -14195.637} C_VEL
LIN {X 0,Y 340.74,Z 274.854,A -85,B 0,C 180,E1 -14199.472,E2 -14199.472} C_VEL
LIN {X 0,Y 340.802,Z 274.843,A -85,B 0,C 180,E1 -14201.979,E2 -14201.979} C_VEL
LIN {X 0,Y 340.879,Z 274.834,A -85,B 0,C 180,E1 -14205.704,E2 -14205.704} C_VEL
LIN {X 0,Y 340.856,Z 274.839,A -85,B 0,C 180,E1 -14209.304,E2 -14209.304} C_VEL
LIN {X 0,Y 341.053,Z 274.817,A -85,B 0,C 180,E1 -14212.896,E2 -14212.896} C_VEL
LIN {X 0,Y 341.174,Z 274.797,A -85,B 0,C 180,E1 -14217.637,E2 -14217.637} C_VEL
LIN {X 0,Y 341.282,Z 274.784,A -85,B 0,C 180,E1 -14219.998,E2 -14219.998} C_VEL
LIN {X 0,Y 341.176,Z 274.801,A -85,B 0,C 180,E1 -14222.359,E2 -14222.359} C_VEL
LIN {X 0,Y 341.08,Z 274.809,A -85,B 0,C 180,E1 -14227.099,E2 -14227.099} C_VEL
LIN {X 0,Y 340.875,Z 274.836,A -85,B 0,C 180,E1 -14230.691,E2 -14230.691} C_VEL
LIN {X 0,Y 340.866,Z 274.84,A -85,B 0,C 180,E1 -14234.322,E2 -14234.322} C_VEL
LIN {X 0,Y 340.839,Z 274.841,A -85,B 0,C 180,E1 -14238.464,E2 -14238.464} C_VEL
LIN {X 0,Y 340.755,Z 274.854,A -85,B 0,C 180,E1 -14241.854,E2 -14241.854} C_VEL
LIN {X 0,Y 340.771,Z 274.851,A -85,B 0,C 180,E1 -14245.661,E2 -14245.661} C_VEL
LIN {X 0,Y 340.727,Z 274.854,A -85,B 0,C 180,E1 -14248.318,E2 -14248.318} C_VEL
LIN {X 0,Y 340.695,Z 274.857,A -85,B 0,C 180,E1 -14251.042,E2 -14251.042} C_VEL
LIN {X 0,Y 340.715,Z 274.857,A -85,B 0,C 180,E1 -14255.276,E2 -14255.276} C_VEL
LIN {X 0,Y 340.714,Z 274.854,A -85,B 0,C 180,E1 -14258.385,E2 -14258.385} C_VEL
LIN {X 0,Y 340.72,Z 274.858,A -85,B 0,C 180,E1 -14261.301,E2 -14261.301} C_VEL
LIN {X 0,Y 340.774,Z 274.847,A -85,B 0,C 180,E1 -14264.519,E2 -14264.519} C_VEL
LIN {X 0,Y 340.743,Z 274.851,A -85,B 0,C 180,E1 -14267.942,E2 -14267.942} C_VEL
LIN {X 0,Y 340.725,Z 274.853,A -85,B 0,C 180,E1 -14270.25,E2 -14270.25} C_VEL
LIN {X 0,Y 340.7,Z 274.857,A -85,B 0,C 180,E1 -14273.556,E2 -14273.556} C_VEL
LIN {X 0,Y 340.681,Z 274.858,A -85,B 0,C 180,E1 -14276.151,E2 -14276.151} C_VEL
LIN {X 0,Y 340.763,Z 274.85,A -85,B 0,C 180,E1 -14280.33,E2 -14280.33} C_VEL
LIN {X 0,Y 340.792,Z 274.847,A -85,B 0,C 180,E1 -14283.017,E2 -14283.017} C_VEL
LIN {X 0,Y 340.75,Z 274.85,A -85,B 0,C 180,E1 -14285.636,E2 -14285.636} C_VEL
LIN {X 0,Y 340.722,Z 274.853,A -85,B 0,C 180,E1 -14289.471,E2 -14289.471} C_VEL
LIN {X 0,Y 340.645,Z 274.864,A -85,B 0,C 180,E1 -14291.971,E2 -14291.971} C_VEL
LIN {X 0,Y 340.143,Z 274.93,A -85,B 0,C 180,E1 -14296.18,E2 -14296.18} C_VEL
LIN {X 0,Y 340.082,Z 275.224,A -85,B 0,C 180,E1 -14296.859,E2 -14296.859} C_VEL
LIN {X 0,Y 339.884,Z 279.039,A -85,B 0,C 180,E1 -14300.477,E2 -14300.477} C_VEL
LIN {X 0,Y 339.99,Z 281.597,A -85,B 0,C 180,E1 -14302.874,E2 -14302.874} C_VEL
LIN {X 0,Y 339.817,Z 285.491,A -85,B 0,C 180,E1 -14306.441,E2 -14306.441} C_VEL
LIN {X 0,Y 339.675,Z 287.724,A -85,B 0,C 180,E1 -14308.442,E2 -14308.442} C_VEL
LIN {X 0,Y 341.319,Z 298.67,A -85,B 0,C 180,E1 -14309.04,E2 -14309.04} C_VEL
LIN {X 0,Y 342.724,Z 307.709,A -85,B 0,C 180,E1 -14309.705,E2 -14309.705} C_VEL
LIN {X 0,Y 342.93,Z 311.278,A -85,B 0,C 180,E1 -14309.998,E2 -14309.998} C_VEL
LIN {X 0,Y 342.244,Z 321.921,A -85,B 0,C 180,E1 -14311.028,E2 -14311.028} C_VEL
LIN {X 0,Y 341.671,Z 330.151,A -85,B 0,C 180,E1 -14312.061,E2 -14312.061} C_VEL
LIN {X 0,Y 341.076,Z 337.804,A -85,B 0,C 180,E1 -14313.247,E2 -14313.247} C_VEL
LIN {X 0,Y 340.596,Z 344.09,A -85,B 0,C 180,E1 -14314.436,E2 -14314.436} C_VEL
LIN {X 0,Y 340.209,Z 349.312,A -85,B 0,C 180,E1 -14315.63,E2 -14315.63} C_VEL
LIN {X 0,Y 340.046,Z 352.562,A -85,B 0,C 180,E1 -14316.486,E2 -14316.486} C_VEL
LIN {X 0,Y 339.728,Z 356.503,A -85,B 0,C 180,E1 -14317.726,E2 -14317.726} C_VEL
LIN {X 0,Y 339.355,Z 360.84,A -85,B 0,C 180,E1 -14319.535,E2 -14319.535} C_VEL
LIN {X 0,Y 339.186,Z 363.05,A -85,B 0,C 180,E1 -14320.746,E2 -14320.746} C_VEL
LIN {X 0,Y 339.119,Z 364.69,A -85,B 0,C 180,E1 -14321.959,E2 -14321.959} C_VEL
LIN {X 0,Y 339.073,Z 365.722,A -85,B 0,C 180,E1 -14323.178,E2 -14323.178} C_VEL
LIN {X 0,Y 339.064,Z 366.241,A -85,B 0,C 180,E1 -14324.401,E2 -14324.401} C_VEL
LIN {X 0,Y 339.11,Z 366.269,A -85,B 0,C 180,E1 -14325.628,E2 -14325.628} C_VEL
LIN {X 0,Y 339.27,Z 365.799,A -85,B 0,C 180,E1 -14326.857,E2 -14326.857} C_VEL
LIN {X 0,Y 339.475,Z 364.799,A -85,B 0,C 180,E1 -14328.09,E2 -14328.09} C_VEL
LIN {X 0,Y 339.924,Z 362.131,A -85,B 0,C 180,E1 -14329.945,E2 -14329.945} C_VEL
LIN {X 0,Y 340.326,Z 359.726,A -85,B 0,C 180,E1 -14331.161,E2 -14331.161} C_VEL
LIN {X 0,Y 340.752,Z 356.517,A -85,B 0,C 180,E1 -14332.429,E2 -14332.429} C_VEL
LIN {X 0,Y 341.51,Z 351.463,A -85,B 0,C 180,E1 -14333.979,E2 -14333.979} C_VEL
LIN {X 0,Y 342.44,Z 344.987,A -85,B 0,C 180,E1 -14335.528,E2 -14335.528} C_VEL
LIN {X 0,Y 343.194,Z 338.561,A -85,B 0,C 180,E1 -14336.775,E2 -14336.775} C_VEL
LIN {X 0,Y 344.103,Z 331.759,A -85,B 0,C 180,E1 -14337.851,E2 -14337.851} C_VEL
LIN {X 0,Y 345.129,Z 323.148,A -85,B 0,C 180,E1 -14338.96,E2 -14338.96} C_VEL
LIN {X 0,Y 345.838,Z 315.079,A -85,B 0,C 180,E1 -14339.797,E2 -14339.797} C_VEL
LIN {X 0,Y 344.155,Z 304.947,A -85,B 0,C 180,E1 -14340.778,E2 -14340.778} C_VEL
LIN {X 0,Y 341.33,Z 294.005,A -85,B 0,C 180,E1 -14341.633,E2 -14341.633} C_VEL
LIN {X 0,Y 339.71,Z 288.312,A -85,B 0,C 180,E1 -14342.049,E2 -14342.049} C_VEL
LIN {X 0,Y 339.836,Z 284.921,A -85,B 0,C 180,E1 -14345.382,E2 -14345.382} C_VEL
LIN {X 0,Y 340.051,Z 282.032,A -85,B 0,C 180,E1 -14348.315,E2 -14348.315} C_VEL
LIN {X 0,Y 340.326,Z 278.475,A -85,B 0,C 180,E1 -14351.98,E2 -14351.98} C_VEL
LIN {X 0,Y 340.467,Z 275.284,A -85,B 0,C 180,E1 -14355.43,E2 -14355.43} C_VEL
LIN {X 0,Y 340.538,Z 274.876,A -85,B 0,C 180,E1 -14357.078,E2 -14357.078} C_VEL
LIN {X 0,Y 340.674,Z 274.862,A -85,B 0,C 180,E1 -14360.248,E2 -14360.248} C_VEL
LIN {X 0,Y 340.686,Z 274.863,A -85,B 0,C 180,E1 -14361.524,E2 -14361.524} C_VEL
LIN {X 0,Y 340.063,Z 274.945,A -85,B 0,C 180,E1 -14362.511,E2 -14362.511} C_VEL
LIN {X 0,Y 337.18,Z 275.301,A -85,B 0,C 180,E1 -14364.115,E2 -14364.115} C_VEL
LIN {X 0,Y 334.72,Z 275.606,A -85,B 0,C 180,E1 -14365.414,E2 -14365.414} C_VEL
LIN {X 0,Y 333.686,Z 275.733,A -85,B 0,C 180,E1 -14366.42,E2 -14366.42} C_VEL
LIN {X 0,Y 333.616,Z 275.742,A -85,B 0,C 180,E1 -14366.761,E2 -14366.761} C_VEL
LIN {X 0,Y 333.676,Z 275.734,A -85,B 0,C 180,E1 -14369.714,E2 -14369.714} C_VEL
LIN {X 0,Y 333.722,Z 275.73,A -85,B 0,C 180,E1 -14372.402,E2 -14372.402} C_VEL
LIN {X 0,Y 333.709,Z 275.731,A -85,B 0,C 180,E1 -14375.092,E2 -14375.092} C_VEL
LIN {X 0,Y 333.66,Z 275.732,A -85,B 0,C 180,E1 -14379.021,E2 -14379.021} C_VEL
LIN {X 0,Y 333.779,Z 275.72,A -85,B 0,C 180,E1 -14381.591,E2 -14381.591} C_VEL
LIN {X 0,Y 333.794,Z 275.714,A -85,B 0,C 180,E1 -14385.579,E2 -14385.579} C_VEL
LIN {X 0,Y 333.824,Z 275.713,A -85,B 0,C 180,E1 -14389.08,E2 -14389.08} C_VEL
LIN {X 0,Y 333.955,Z 275.697,A -85,B 0,C 180,E1 -14392.748,E2 -14392.748} C_VEL
LIN {X 0,Y 333.795,Z 275.718,A -85,B 0,C 180,E1 -14395.171,E2 -14395.171} C_VEL
LIN {X 0,Y 334.096,Z 275.677,A -85,B 0,C 180,E1 -14397.591,E2 -14397.591} C_VEL
LIN {X 0,Y 334.235,Z 275.664,A -85,B 0,C 180,E1 -14400.002,E2 -14400.002} C_VEL
LIN {X 0,Y 334.094,Z 275.678,A -85,B 0,C 180,E1 -14402.413,E2 -14402.413} C_VEL
LIN {X 0,Y 334.016,Z 275.692,A -85,B 0,C 180,E1 -14407.255,E2 -14407.255} C_VEL
LIN {X 0,Y 333.827,Z 275.714,A -85,B 0,C 180,E1 -14410.924,E2 -14410.924} C_VEL
LIN {X 0,Y 333.8,Z 275.719,A -85,B 0,C 180,E1 -14414.637,E2 -14414.637} C_VEL
LIN {X 0,Y 333.789,Z 275.719,A -85,B 0,C 180,E1 -14418.657,E2 -14418.657} C_VEL
LIN {X 0,Y 333.647,Z 275.737,A -85,B 0,C 180,E1 -14422.283,E2 -14422.283} C_VEL
LIN {X 0,Y 333.694,Z 275.733,A -85,B 0,C 180,E1 -14425.096,E2 -14425.096} C_VEL
LIN {X 0,Y 333.649,Z 275.742,A -85,B 0,C 180,E1 -14428.98,E2 -14428.98} C_VEL
LIN {X 0,Y 333.638,Z 275.744,A -85,B 0,C 180,E1 -14432.589,E2 -14432.589} C_VEL
LIN {X 0,Y 333.672,Z 275.738,A -85,B 0,C 180,E1 -14436.141,E2 -14436.141} C_VEL
LIN {X 0,Y 333.667,Z 275.737,A -85,B 0,C 180,E1 -14439.191,E2 -14439.191} C_VEL
LIN {X 0,Y 333.663,Z 275.737,A -85,B 0,C 180,E1 -14442.509,E2 -14442.509} C_VEL
LIN {X 0,Y 333.619,Z 275.804,A -85,B 0,C 180,E1 -14446.263,E2 -14446.263} C_VEL
LIN {X 0,Y 334.409,Z 279.695,A -85,B 0,C 180,E1 -14449.348,E2 -14449.348} C_VEL
LIN {X 0,Y 335.167,Z 284.415,A -85,B 0,C 180,E1 -14452.828,E2 -14452.828} C_VEL
LIN {X 0,Y 335.727,Z 288.408,A -85,B 0,C 180,E1 -14455.585,E2 -14455.585} C_VEL
LIN {X 0,Y 335.79,Z 290.632,A -85,B 0,C 180,E1 -14457.034,E2 -14457.034} C_VEL
LIN {X 0,Y 334.931,Z 296.239,A -85,B 0,C 180,E1 -14460.457,E2 -14460.457} C_VEL
LIN {X 0,Y 334.137,Z 301.882,A -85,B 0,C 180,E1 -14463.79,E2 -14463.79} C_VEL
LIN {X 0,Y 333.33,Z 308.72,A -85,B 0,C 180,E1 -14467.698,E2 -14467.698} C_VEL
LIN {X 0,Y 332.822,Z 315.552,A -85,B 0,C 180,E1 -14471.516,E2 -14471.516} C_VEL
LIN {X 0,Y 335.028,Z 326.933,A -85,B 0,C 180,E1 -14472.198,E2 -14472.198} C_VEL
LIN {X 0,Y 336.453,Z 337.098,A -85,B 0,C 180,E1 -14472.998,E2 -14472.998} C_VEL
LIN {X 0,Y 337.12,Z 344.858,A -85,B 0,C 180,E1 -14473.725,E2 -14473.725} C_VEL
LIN {X 0,Y 337.143,Z 352.771,A -85,B 0,C 180,E1 -14474.588,E2 -14474.588} C_VEL
LIN {X 0,Y 336.281,Z 360.895,A -85,B 0,C 180,E1 -14475.632,E2 -14475.632} C_VEL
LIN {X 0,Y 335.283,Z 367.632,A -85,B 0,C 180,E1 -14476.671,E2 -14476.671} C_VEL
LIN {X 0,Y 334.428,Z 374.033,A -85,B 0,C 180,E1 -14477.871,E2 -14477.871} C_VEL
LIN {X 0,Y 333.706,Z 379.371,A -85,B 0,C 180,E1 -14479.076,E2 -14479.076} C_VEL
LIN {X 0,Y 333.108,Z 383.842,A -85,B 0,C 180,E1 -14480.284,E2 -14480.284} C_VEL
LIN {X 0,Y 332.655,Z 387.582,A -85,B 0,C 180,E1 -14481.497,E2 -14481.497} C_VEL
LIN {X 0,Y 332.249,Z 391.857,A -85,B 0,C 180,E1 -14483.321,E2 -14483.321} C_VEL
LIN {X 0,Y 332.051,Z 394.877,A -85,B 0,C 180,E1 -14485.145,E2 -14485.145} C_VEL
LIN {X 0,Y 332.04,Z 396.24,A -85,B 0,C 180,E1 -14486.361,E2 -14486.361} C_VEL
LIN {X 0,Y 331.988,Z 397.13,A -85,B 0,C 180,E1 -14487.575,E2 -14487.575} C_VEL
LIN {X 0,Y 332.062,Z 397.479,A -85,B 0,C 180,E1 -14488.789,E2 -14488.789} C_VEL
LIN {X 0,Y 332.135,Z 397.268,A -85,B 0,C 180,E1 -14490.002,E2 -14490.002} C_VEL
LIN {X 0,Y 332.108,Z 396.587,A -85,B 0,C 180,E1 -14491.214,E2 -14491.214} C_VEL
LIN {X 0,Y 332.03,Z 395.424,A -85,B 0,C 180,E1 -14492.428,E2 -14492.428} C_VEL
LIN {X 0,Y 332.135,Z 392.612,A -85,B 0,C 180,E1 -14494.249,E2 -14494.249} C_VEL
LIN {X 0,Y 332.146,Z 388.507,A -85,B 0,C 180,E1 -14496.075,E2 -14496.075} C_VEL
LIN {X 0,Y 332.455,Z 382.945,A -85,B 0,C 180,E1 -14497.899,E2 -14497.899} C_VEL
LIN {X 0,Y 332.805,Z 376.822,A -85,B 0,C 180,E1 -14499.421,E2 -14499.421} C_VEL
LIN {X 0,Y 333.24,Z 370.844,A -85,B 0,C 180,E1 -14500.636,E2 -14500.636} C_VEL
LIN {X 0,Y 333.753,Z 363.555,A -85,B 0,C 180,E1 -14501.849,E2 -14501.849} C_VEL
LIN {X 0,Y 334.448,Z 355.785,A -85,B 0,C 180,E1 -14502.903,E2 -14502.903} C_VEL
LIN {X 0,Y 334.883,Z 349.128,A -85,B 0,C 180,E1 -14503.654,E2 -14503.654} C_VEL
LIN {X 0,Y 334.435,Z 340.744,A -85,B 0,C 180,E1 -14504.452,E2 -14504.452} C_VEL
LIN {X 0,Y 333.814,Z 332.463,A -85,B 0,C 180,E1 -14505.087,E2 -14505.087} C_VEL
LIN {X 0,Y 333.014,Z 322.88,A -85,B 0,C 180,E1 -14505.65,E2 -14505.65} C_VEL
LIN {X 0,Y 332.345,Z 316.139,A -85,B 0,C 180,E1 -14505.958,E2 -14505.958} C_VEL
LIN {X 0,Y 332.673,Z 309.04,A -85,B 0,C 180,E1 -14509.757,E2 -14509.757} C_VEL
LIN {X 0,Y 333.118,Z 303.073,A -85,B 0,C 180,E1 -14512.975,E2 -14512.975} C_VEL
LIN {X 0,Y 333.787,Z 295.882,A -85,B 0,C 180,E1 -14516.918,E2 -14516.918} C_VEL
LIN {X 0,Y 334.527,Z 289.435,A -85,B 0,C 180,E1 -14520.528,E2 -14520.528} C_VEL
LIN {X 0,Y 335.032,Z 285.043,A -85,B 0,C 180,E1 -14523.054,E2 -14523.054} C_VEL
LIN {X 0,Y 334.799,Z 281.734,A -85,B 0,C 180,E1 -14525.046,E2 -14525.046} C_VEL
LIN {X 0,Y 333.724,Z 275.727,A -85,B 0,C 180,E1 -14528.89,E2 -14528.89} C_VEL
LIN {X 0,Y 333.642,Z 275.736,A -85,B 0,C 180,E1 -14532.5,E2 -14532.5} C_VEL
LIN {X 0,Y 333.607,Z 275.745,A -85,B 0,C 180,E1 -14535.955,E2 -14535.955} C_VEL
LIN {X 0,Y 333.658,Z 275.734,A -85,B 0,C 180,E1 -14539.315,E2 -14539.315} C_VEL
LIN {X 0,Y 333.675,Z 275.732,A -85,B 0,C 180,E1 -14543.168,E2 -14543.168} C_VEL
LIN {X 0,Y 333.684,Z 275.732,A -85,B 0,C 180,E1 -14545.341,E2 -14545.341} C_VEL
LIN {X 0,Y 333.713,Z 275.73,A -85,B 0,C 180,E1 -14549.71,E2 -14549.71} C_VEL
LIN {X 0,Y 333.754,Z 275.721,A -85,B 0,C 180,E1 -14552.4,E2 -14552.4} C_VEL
LIN {X 0,Y 333.736,Z 275.726,A -85,B 0,C 180,E1 -14555.09,E2 -14555.09} C_VEL
LIN {X 0,Y 333.68,Z 275.734,A -85,B 0,C 180,E1 -14559.017,E2 -14559.017} C_VEL
LIN {X 0,Y 333.75,Z 275.723,A -85,B 0,C 180,E1 -14561.585,E2 -14561.585} C_VEL
LIN {X 0,Y 333.818,Z 275.714,A -85,B 0,C 180,E1 -14565.575,E2 -14565.575} C_VEL
LIN {X 0,Y 333.826,Z 275.716,A -85,B 0,C 180,E1 -14569.076,E2 -14569.076} C_VEL
LIN {X 0,Y 334,Z 275.695,A -85,B 0,C 180,E1 -14572.745,E2 -14572.745} C_VEL
LIN {X 0,Y 333.812,Z 275.716,A -85,B 0,C 180,E1 -14575.167,E2 -14575.167} C_VEL
LIN {X 0,Y 334.111,Z 275.676,A -85,B 0,C 180,E1 -14577.587,E2 -14577.587} C_VEL
LIN {X 0,Y 334.234,Z 275.662,A -85,B 0,C 180,E1 -14579.998,E2 -14579.998} C_VEL
LIN {X 0,Y 334.113,Z 275.681,A -85,B 0,C 180,E1 -14582.409,E2 -14582.409} C_VEL
LIN {X 0,Y 334.03,Z 275.686,A -85,B 0,C 180,E1 -14587.25,E2 -14587.25} C_VEL
LIN {X 0,Y 333.838,Z 275.711,A -85,B 0,C 180,E1 -14590.919,E2 -14590.919} C_VEL
LIN {X 0,Y 333.811,Z 275.715,A -85,B 0,C 180,E1 -14594.632,E2 -14594.632} C_VEL
LIN {X 0,Y 333.798,Z 275.716,A -85,B 0,C 180,E1 -14598.652,E2 -14598.652} C_VEL
LIN {X 0,Y 333.693,Z 275.731,A -85,B 0,C 180,E1 -14602.275,E2 -14602.275} C_VEL
LIN {X 0,Y 333.734,Z 275.725,A -85,B 0,C 180,E1 -14606.243,E2 -14606.243} C_VEL
LIN {X 0,Y 333.688,Z 275.729,A -85,B 0,C 180,E1 -14608.971,E2 -14608.971} C_VEL
LIN {X 0,Y 333.64,Z 275.735,A -85,B 0,C 180,E1 -14612.584,E2 -14612.584} C_VEL
LIN {X 0,Y 333.673,Z 275.732,A -85,B 0,C 180,E1 -14616.136,E2 -14616.136} C_VEL
LIN {X 0,Y 333.679,Z 275.733,A -85,B 0,C 180,E1 -14619.184,E2 -14619.184} C_VEL
LIN {X 0,Y 333.697,Z 275.728,A -85,B 0,C 180,E1 -14622.51,E2 -14622.51} C_VEL
LIN {X 0,Y 333.721,Z 275.725,A -85,B 0,C 180,E1 -14625.974,E2 -14625.974} C_VEL
LIN {X 0,Y 333.693,Z 275.733,A -85,B 0,C 180,E1 -14629.302,E2 -14629.302} C_VEL
LIN {X 0,Y 333.656,Z 275.737,A -85,B 0,C 180,E1 -14633.165,E2 -14633.165} C_VEL
LIN {X 0,Y 333.663,Z 275.734,A -85,B 0,C 180,E1 -14635.338,E2 -14635.338} C_VEL
LIN {X 0,Y 333.691,Z 275.729,A -85,B 0,C 180,E1 -14639.708,E2 -14639.708} C_VEL
LIN {X 0,Y 333.732,Z 275.726,A -85,B 0,C 180,E1 -14642.399,E2 -14642.399} C_VEL
LIN {X 0,Y 333.719,Z 275.727,A -85,B 0,C 180,E1 -14645.089,E2 -14645.089} C_VEL
LIN {X 0,Y 333.67,Z 275.733,A -85,B 0,C 180,E1 -14649.017,E2 -14649.017} C_VEL
LIN {X 0,Y 333.597,Z 275.74,A -85,B 0,C 180,E1 -14651.577,E2 -14651.577} C_VEL
LIN {X 0,Y 333.189,Z 275.792,A -85,B 0,C 180,E1 -14655.336,E2 -14655.336} C_VEL
LIN {X 0,Y 333.039,Z 275.817,A -85,B 0,C 180,E1 -14656.576,E2 -14656.576} C_VEL
LIN {X 0,Y 332.828,Z 279.521,A -85,B 0,C 180,E1 -14660.273,E2 -14660.273} C_VEL
LIN {X 0,Y 332.93,Z 282.147,A -85,B 0,C 180,E1 -14662.788,E2 -14662.788} C_VEL
LIN {X 0,Y 332.763,Z 286.04,A -85,B 0,C 180,E1 -14666.366,E2 -14666.366} C_VEL
LIN {X 0,Y 332.601,Z 288.043,A -85,B 0,C 180,E1 -14668.182,E2 -14668.182} C_VEL
LIN {X 0,Y 334.41,Z 299.954,A -85,B 0,C 180,E1 -14668.869,E2 -14668.869} C_VEL
LIN {X 0,Y 335.776,Z 308.805,A -85,B 0,C 180,E1 -14669.549,E2 -14669.549} C_VEL
LIN {X 0,Y 335.846,Z 314.086,A -85,B 0,C 180,E1 -14669.998,E2 -14669.998} C_VEL
LIN {X 0,Y 335.107,Z 324.015,A -85,B 0,C 180,E1 -14671.05,E2 -14671.05} C_VEL
LIN {X 0,Y 334.534,Z 331.948,A -85,B 0,C 180,E1 -14672.105,E2 -14672.105} C_VEL
LIN {X 0,Y 333.958,Z 339.355,A -85,B 0,C 180,E1 -14673.316,E2 -14673.316} C_VEL
LIN {X 0,Y 333.353,Z 346.866,A -85,B 0,C 180,E1 -14674.836,E2 -14674.836} C_VEL
LIN {X 0,Y 332.979,Z 352.927,A -85,B 0,C 180,E1 -14676.417,E2 -14676.417} C_VEL
LIN {X 0,Y 332.584,Z 357.396,A -85,B 0,C 180,E1 -14677.893,E2 -14677.893} C_VEL
LIN {X 0,Y 332.361,Z 360.411,A -85,B 0,C 180,E1 -14679.124,E2 -14679.124} C_VEL
LIN {X 0,Y 332.084,Z 363.678,A -85,B 0,C 180,E1 -14680.978,E2 -14680.978} C_VEL
LIN {X 0,Y 332.016,Z 365.232,A -85,B 0,C 180,E1 -14682.219,E2 -14682.219} C_VEL
LIN {X 0,Y 331.975,Z 366.228,A -85,B 0,C 180,E1 -14683.465,E2 -14683.465} C_VEL
LIN {X 0,Y 331.992,Z 366.635,A -85,B 0,C 180,E1 -14684.714,E2 -14684.714} C_VEL
LIN {X 0,Y 332.05,Z 366.546,A -85,B 0,C 180,E1 -14685.969,E2 -14685.969} C_VEL
LIN {X 0,Y 332.371,Z 365.419,A -85,B 0,C 180,E1 -14687.923,E2 -14687.923} C_VEL
LIN {X 0,Y 332.793,Z 363.191,A -85,B 0,C 180,E1 -14689.747,E2 -14689.747} C_VEL
LIN {X 0,Y 333.365,Z 359.779,A -85,B 0,C 180,E1 -14691.511,E2 -14691.511} C_VEL
LIN {X 0,Y 333.91,Z 356.18,A -85,B 0,C 180,E1 -14692.914,E2 -14692.914} C_VEL
LIN {X 0,Y 334.726,Z 350.933,A -85,B 0,C 180,E1 -14694.497,E2 -14694.497} C_VEL
LIN {X 0,Y 335.512,Z 345.778,A -85,B 0,C 180,E1 -14695.754,E2 -14695.754} C_VEL
LIN {X 0,Y 336.317,Z 339.408,A -85,B 0,C 180,E1 -14697.031,E2 -14697.031} C_VEL
LIN {X 0,Y 337.285,Z 332.714,A -85,B 0,C 180,E1 -14698.126,E2 -14698.126} C_VEL
LIN {X 0,Y 338.202,Z 325.582,A -85,B 0,C 180,E1 -14699.09,E2 -14699.09} C_VEL
LIN {X 0,Y 338.989,Z 317.81,A -85,B 0,C 180,E1 -14699.957,E2 -14699.957} C_VEL
LIN {X 0,Y 338.748,Z 313.263,A -85,B 0,C 180,E1 -14700.444,E2 -14700.444} C_VEL
LIN {X 0,Y 336.67,Z 303.007,A -85,B 0,C 180,E1 -14701.415,E2 -14701.415} C_VEL
LIN {X 0,Y 334.061,Z 293.518,A -85,B 0,C 180,E1 -14702.171,E2 -14702.171} C_VEL
LIN {X 0,Y 332.697,Z 288.673,A -85,B 0,C 180,E1 -14702.538,E2 -14702.538} C_VEL
LIN {X 0,Y 332.883,Z 284.57,A -85,B 0,C 180,E1 -14706.657,E2 -14706.657} C_VEL
LIN {X 0,Y 333.178,Z 280.798,A -85,B 0,C 180,E1 -14710.595,E2 -14710.595} C_VEL
LIN {X 0,Y 333.392,Z 277.558,A -85,B 0,C 180,E1 -14714.076,E2 -14714.076} C_VEL
LIN {X 0,Y 333.426,Z 275.904,A -85,B 0,C 180,E1 -14715.931,E2 -14715.931} C_VEL
LIN {X 0,Y 333.584,Z 275.747,A -85,B 0,C 180,E1 -14719.325,E2 -14719.325} C_VEL
LIN {X 0,Y 333.635,Z 275.742,A -85,B 0,C 180,E1 -14722.35,E2 -14722.35} C_VEL
LIN {X 0,Y 333.655,Z 275.738,A -85,B 0,C 180,E1 -14725.343,E2 -14725.343} C_VEL
LIN {X 0,Y 333.616,Z 275.742,A -85,B 0,C 180,E1 -14726.761,E2 -14726.761} C_VEL
LIN {X 0,Y 332.993,Z 275.825,A -85,B 0,C 180,E1 -14727.769,E2 -14727.769} C_VEL
LIN {X 0,Y 330.177,Z 276.179,A -85,B 0,C 180,E1 -14729.411,E2 -14729.411} C_VEL
LIN {X 0,Y 327.763,Z 276.476,A -85,B 0,C 180,E1 -14730.74,E2 -14730.74} C_VEL
LIN {X 0,Y 326.72,Z 276.6,A -85,B 0,C 180,E1 -14731.769,E2 -14731.769} C_VEL
LIN {X 0,Y 326.632,Z 276.61,A -85,B 0,C 180,E1 -14732.117,E2 -14732.117} C_VEL
LIN {X 0,Y 326.671,Z 276.606,A -85,B 0,C 180,E1 -14734.629,E2 -14734.629} C_VEL
LIN {X 0,Y 326.605,Z 276.613,A -85,B 0,C 180,E1 -14738.545,E2 -14738.545} C_VEL
LIN {X 0,Y 326.729,Z 276.599,A -85,B 0,C 180,E1 -14741.179,E2 -14741.179} C_VEL
LIN {X 0,Y 326.749,Z 276.592,A -85,B 0,C 180,E1 -14745.435,E2 -14745.435} C_VEL
LIN {X 0,Y 326.76,Z 276.593,A -85,B 0,C 180,E1 -14748.841,E2 -14748.841} C_VEL
LIN {X 0,Y 326.909,Z 276.576,A -85,B 0,C 180,E1 -14752.591,E2 -14752.591} C_VEL
LIN {X 0,Y 326.761,Z 276.594,A -85,B 0,C 180,E1 -14755.067,E2 -14755.067} C_VEL
LIN {X 0,Y 327.037,Z 276.556,A -85,B 0,C 180,E1 -14757.539,E2 -14757.539} C_VEL
LIN {X 0,Y 327.187,Z 276.542,A -85,B 0,C 180,E1 -14760.002,E2 -14760.002} C_VEL
LIN {X 0,Y 327.035,Z 276.557,A -85,B 0,C 180,E1 -14762.466,E2 -14762.466} C_VEL
LIN {X 0,Y 326.987,Z 276.561,A -85,B 0,C 180,E1 -14766.171,E2 -14766.171} C_VEL
LIN {X 0,Y 326.905,Z 276.579,A -85,B 0,C 180,E1 -14768.657,E2 -14768.657} C_VEL
LIN {X 0,Y 326.729,Z 276.599,A -85,B 0,C 180,E1 -14772.424,E2 -14772.424} C_VEL
LIN {X 0,Y 326.746,Z 276.598,A -85,B 0,C 180,E1 -14774.96,E2 -14774.96} C_VEL
LIN {X 0,Y 326.725,Z 276.599,A -85,B 0,C 180,E1 -14778.84,E2 -14778.84} C_VEL
LIN {X 0,Y 326.593,Z 276.619,A -85,B 0,C 180,E1 -14782.791,E2 -14782.791} C_VEL
LIN {X 0,Y 326.633,Z 276.613,A -85,B 0,C 180,E1 -14785.49,E2 -14785.49} C_VEL
LIN {X 0,Y 326.611,Z 276.618,A -85,B 0,C 180,E1 -14789.666,E2 -14789.666} C_VEL
LIN {X 0,Y 326.612,Z 276.619,A -85,B 0,C 180,E1 -14792.948,E2 -14792.948} C_VEL
LIN {X 0,Y 326.608,Z 276.62,A -85,B 0,C 180,E1 -14795.522,E2 -14795.522} C_VEL
LIN {X 0,Y 326.629,Z 276.614,A -85,B 0,C 180,E1 -14799.234,E2 -14799.234} C_VEL
LIN {X 0,Y 326.596,Z 276.619,A -85,B 0,C 180,E1 -14802.979,E2 -14802.979} C_VEL
LIN {X 0,Y 326.563,Z 276.661,A -85,B 0,C 180,E1 -14805.735,E2 -14805.735} C_VEL
LIN {X 0,Y 327.268,Z 280.319,A -85,B 0,C 180,E1 -14808.733,E2 -14808.733} C_VEL
LIN {X 0,Y 328.118,Z 285.148,A -85,B 0,C 180,E1 -14812.423,E2 -14812.423} C_VEL
LIN {X 0,Y 328.728,Z 289.49,A -85,B 0,C 180,E1 -14815.492,E2 -14815.492} C_VEL
LIN {X 0,Y 328.615,Z 292.807,A -85,B 0,C 180,E1 -14817.681,E2 -14817.681} C_VEL
LIN {X 0,Y 327.889,Z 297.276,A -85,B 0,C 180,E1 -14820.465,E2 -14820.465} C_VEL
LIN {X 0,Y 326.935,Z 304.045,A -85,B 0,C 180,E1 -14824.539,E2 -14824.539} C_VEL
LIN {X 0,Y 326.101,Z 310.862,A -85,B 0,C 180,E1 -14828.51,E2 -14828.51} C_VEL
LIN {X 0,Y 325.802,Z 315.176,A -85,B 0,C 180,E1 -14830.985,E2 -14830.985} C_VEL
LIN {X 0,Y 328.266,Z 327.546,A -85,B 0,C 180,E1 -14831.785,E2 -14831.785} C_VEL
LIN {X 0,Y 329.653,Z 337.821,A -85,B 0,C 180,E1 -14832.636,E2 -14832.636} C_VEL
LIN {X 0,Y 330.295,Z 345.555,A -85,B 0,C 180,E1 -14833.399,E2 -14833.399} C_VEL
LIN {X 0,Y 330.305,Z 353.121,A -85,B 0,C 180,E1 -14834.261,E2 -14834.261} C_VEL
LIN {X 0,Y 329.438,Z 361.129,A -85,B 0,C 180,E1 -14835.327,E2 -14835.327} C_VEL
LIN {X 0,Y 328.387,Z 367.773,A -85,B 0,C 180,E1 -14836.386,E2 -14836.386} C_VEL
LIN {X 0,Y 327.48,Z 374.095,A -85,B 0,C 180,E1 -14837.609,E2 -14837.609} C_VEL
LIN {X 0,Y 326.729,Z 379.364,A -85,B 0,C 180,E1 -14838.839,E2 -14838.839} C_VEL
LIN {X 0,Y 326.113,Z 383.775,A -85,B 0,C 180,E1 -14840.074,E2 -14840.074} C_VEL
LIN {X 0,Y 325.432,Z 388.991,A -85,B 0,C 180,E1 -14841.932,E2 -14841.932} C_VEL
LIN {X 0,Y 325.187,Z 391.684,A -85,B 0,C 180,E1 -14843.175,E2 -14843.175} C_VEL
LIN {X 0,Y 325.009,Z 393.405,A -85,B 0,C 180,E1 -14844.111,E2 -14844.111} C_VEL
LIN {X 0,Y 324.966,Z 395.975,A -85,B 0,C 180,E1 -14846.282,E2 -14846.282} C_VEL
LIN {X 0,Y 324.904,Z 396.82,A -85,B 0,C 180,E1 -14847.522,E2 -14847.522} C_VEL
LIN {X 0,Y 324.964,Z 397.161,A -85,B 0,C 180,E1 -14848.762,E2 -14848.762} C_VEL
LIN {X 0,Y 325.043,Z 396.915,A -85,B 0,C 180,E1 -14850.002,E2 -14850.002} C_VEL
LIN {X 0,Y 325.012,Z 396.191,A -85,B 0,C 180,E1 -14851.241,E2 -14851.241} C_VEL
LIN {X 0,Y 324.944,Z 394.984,A -85,B 0,C 180,E1 -14852.481,E2 -14852.481} C_VEL
LIN {X 0,Y 325.041,Z 392.124,A -85,B 0,C 180,E1 -14854.342,E2 -14854.342} C_VEL
LIN {X 0,Y 325.038,Z 388.632,A -85,B 0,C 180,E1 -14855.938,E2 -14855.938} C_VEL
LIN {X 0,Y 325.351,Z 383.363,A -85,B 0,C 180,E1 -14857.761,E2 -14857.761} C_VEL
LIN {X 0,Y 325.744,Z 376.095,A -85,B 0,C 180,E1 -14859.627,E2 -14859.627} C_VEL
LIN {X 0,Y 326.244,Z 370.04,A -85,B 0,C 180,E1 -14860.866,E2 -14860.866} C_VEL
LIN {X 0,Y 326.8,Z 362.655,A -85,B 0,C 180,E1 -14862.105,E2 -14862.105} C_VEL
LIN {X 0,Y 327.401,Z 356.002,A -85,B 0,C 180,E1 -14863.028,E2 -14863.028} C_VEL
LIN {X 0,Y 327.856,Z 349.621,A -85,B 0,C 180,E1 -14863.778,E2 -14863.778} C_VEL
LIN {X 0,Y 327.412,Z 341.053,A -85,B 0,C 180,E1 -14864.626,E2 -14864.626} C_VEL
LIN {X 0,Y 326.718,Z 331.699,A -85,B 0,C 180,E1 -14865.36,E2 -14865.36} C_VEL
LIN {X 0,Y 325.924,Z 322.295,A -85,B 0,C 180,E1 -14865.919,E2 -14865.919} C_VEL
LIN {X 0,Y 325.284,Z 315.833,A -85,B 0,C 180,E1 -14866.233,E2 -14866.233} C_VEL
LIN {X 0,Y 325.633,Z 308.58,A -85,B 0,C 180,E1 -14870.203,E2 -14870.203} C_VEL
LIN {X 0,Y 326.105,Z 302.624,A -85,B 0,C 180,E1 -14873.498,E2 -14873.498} C_VEL
LIN {X 0,Y 326.688,Z 296.649,A -85,B 0,C 180,E1 -14876.859,E2 -14876.859} C_VEL
LIN {X 0,Y 327.577,Z 289.462,A -85,B 0,C 180,E1 -14880.993,E2 -14880.993} C_VEL
LIN {X 0,Y 327.988,Z 285.527,A -85,B 0,C 180,E1 -14883.311,E2 -14883.311} C_VEL
LIN {X 0,Y 327.675,Z 282.15,A -85,B 0,C 180,E1 -14885.408,E2 -14885.408} C_VEL
LIN {X 0,Y 326.684,Z 276.603,A -85,B 0,C 180,E1 -14889.134,E2 -14889.134} C_VEL
LIN {X 0,Y 326.572,Z 276.617,A -85,B 0,C 180,E1 -14893.526,E2 -14893.526} C_VEL
LIN {X 0,Y 326.586,Z 276.614,A -85,B 0,C 180,E1 -14897.028,E2 -14897.028} C_VEL
LIN {X 0,Y 326.621,Z 276.609,A -85,B 0,C 180,E1 -14900.773,E2 -14900.773} C_VEL
LIN {X 0,Y 326.622,Z 276.609,A -85,B 0,C 180,E1 -14904.48,E2 -14904.48} C_VEL
LIN {X 0,Y 326.618,Z 276.614,A -85,B 0,C 180,E1 -14907.455,E2 -14907.455} C_VEL
LIN {X 0,Y 326.671,Z 276.603,A -85,B 0,C 180,E1 -14910.34,E2 -14910.34} C_VEL
LIN {X 0,Y 326.7,Z 276.599,A -85,B 0,C 180,E1 -14914.515,E2 -14914.515} C_VEL
LIN {X 0,Y 326.628,Z 276.609,A -85,B 0,C 180,E1 -14918.542,E2 -14918.542} C_VEL
LIN {X 0,Y 326.673,Z 276.603,A -85,B 0,C 180,E1 -14922.469,E2 -14922.469} C_VEL
LIN {X 0,Y 326.768,Z 276.591,A -85,B 0,C 180,E1 -14926.313,E2 -14926.313} C_VEL
LIN {X 0,Y 326.791,Z 276.588,A -85,B 0,C 180,E1 -14930.091,E2 -14930.091} C_VEL
LIN {X 0,Y 326.989,Z 276.563,A -85,B 0,C 180,E1 -14933.829,E2 -14933.829} C_VEL
LIN {X 0,Y 327.052,Z 276.556,A -85,B 0,C 180,E1 -14937.535,E2 -14937.535} C_VEL
LIN {X 0,Y 327.186,Z 276.54,A -85,B 0,C 180,E1 -14939.998,E2 -14939.998} C_VEL
LIN {X 0,Y 327.053,Z 276.56,A -85,B 0,C 180,E1 -14942.461,E2 -14942.461} C_VEL
LIN {X 0,Y 326.977,Z 276.565,A -85,B 0,C 180,E1 -14946.635,E2 -14946.635} C_VEL
LIN {X 0,Y 326.818,Z 276.587,A -85,B 0,C 180,E1 -14949.904,E2 -14949.904} C_VEL
LIN {X 0,Y 326.762,Z 276.593,A -85,B 0,C 180,E1 -14953.683,E2 -14953.683} C_VEL
LIN {X 0,Y 326.701,Z 276.6,A -85,B 0,C 180,E1 -14957.525,E2 -14957.525} C_VEL
LIN {X 0,Y 326.665,Z 276.608,A -85,B 0,C 180,E1 -14960.132,E2 -14960.132} C_VEL
LIN {X 0,Y 326.652,Z 276.609,A -85,B 0,C 180,E1 -14964.126,E2 -14964.126} C_VEL
LIN {X 0,Y 326.682,Z 276.602,A -85,B 0,C 180,E1 -14966.855,E2 -14966.855} C_VEL
LIN {X 0,Y 326.632,Z 276.608,A -85,B 0,C 180,E1 -14970.607,E2 -14970.607} C_VEL
LIN {X 0,Y 326.603,Z 276.613,A -85,B 0,C 180,E1 -14974.016,E2 -14974.016} C_VEL
LIN {X 0,Y 326.626,Z 276.612,A -85,B 0,C 180,E1 -14977.236,E2 -14977.236} C_VEL
LIN {X 0,Y 326.63,Z 276.608,A -85,B 0,C 180,E1 -14980.199,E2 -14980.199} C_VEL
LIN {X 0,Y 326.651,Z 276.609,A -85,B 0,C 180,E1 -14983.506,E2 -14983.506} C_VEL
LIN {X 0,Y 326.642,Z 276.61,A -85,B 0,C 180,E1 -14987.011,E2 -14987.011} C_VEL
LIN {X 0,Y 326.636,Z 276.61,A -85,B 0,C 180,E1 -14990.763,E2 -14990.763} C_VEL
LIN {X 0,Y 326.602,Z 276.613,A -85,B 0,C 180,E1 -14994.477,E2 -14994.477} C_VEL
LIN {X 0,Y 326.596,Z 276.613,A -85,B 0,C 180,E1 -14997.453,E2 -14997.453} C_VEL
LIN {X 0,Y 326.649,Z 276.607,A -85,B 0,C 180,E1 -15000.338,E2 -15000.338} C_VEL
LIN {X 0,Y 326.679,Z 276.606,A -85,B 0,C 180,E1 -15004.514,E2 -15004.514} C_VEL
LIN {X 0,Y 326.634,Z 276.613,A -85,B 0,C 180,E1 -15008.543,E2 -15008.543} C_VEL
LIN {X 0,Y 326.549,Z 276.618,A -85,B 0,C 180,E1 -15011.247,E2 -15011.247} C_VEL
LIN {X 0,Y 326.169,Z 276.666,A -85,B 0,C 180,E1 -15015.014,E2 -15015.014} C_VEL
LIN {X 0,Y 326.031,Z 276.688,A -85,B 0,C 180,E1 -15016.282,E2 -15016.282} C_VEL
LIN {X 0,Y 325.9,Z 277.464,A -85,B 0,C 180,E1 -15017.545,E2 -15017.545} C_VEL
LIN {X 0,Y 325.762,Z 281.313,A -85,B 0,C 180,E1 -15021.313,E2 -15021.313} C_VEL
LIN {X 0,Y 325.756,Z 283.927,A -85,B 0,C 180,E1 -15023.806,E2 -15023.806} C_VEL
LIN {X 0,Y 325.71,Z 286.562,A -85,B 0,C 180,E1 -15026.287,E2 -15026.287} C_VEL
LIN {X 0,Y 325.537,Z 288.315,A -85,B 0,C 180,E1 -15027.911,E2 -15027.911} C_VEL
LIN {X 0,Y 327.392,Z 300.119,A -85,B 0,C 180,E1 -15028.615,E2 -15028.615} C_VEL
LIN {X 0,Y 328.815,Z 309.89,A -85,B 0,C 180,E1 -15029.386,E2 -15029.386} C_VEL
LIN {X 0,Y 328.838,Z 315.038,A -85,B 0,C 180,E1 -15029.845,E2 -15029.845} C_VEL
LIN {X 0,Y 328.201,Z 323.61,A -85,B 0,C 180,E1 -15030.765,E2 -15030.765} C_VEL
LIN {X 0,Y 327.571,Z 331.674,A -85,B 0,C 180,E1 -15031.843,E2 -15031.843} C_VEL
LIN {X 0,Y 327.108,Z 337.471,A -85,B 0,C 180,E1 -15032.769,E2 -15032.769} C_VEL
LIN {X 0,Y 326.598,Z 343.921,A -85,B 0,C 180,E1 -15034.009,E2 -15034.009} C_VEL
LIN {X 0,Y 326.11,Z 349.295,A -85,B 0,C 180,E1 -15035.254,E2 -15035.254} C_VEL
LIN {X 0,Y 325.976,Z 352.774,A -85,B 0,C 180,E1 -15036.187,E2 -15036.187} C_VEL
LIN {X 0,Y 325.601,Z 356.664,A -85,B 0,C 180,E1 -15037.439,E2 -15037.439} C_VEL
LIN {X 0,Y 325.218,Z 361.163,A -85,B 0,C 180,E1 -15039.326,E2 -15039.326} C_VEL
LIN {X 0,Y 324.964,Z 364.303,A -85,B 0,C 180,E1 -15041.222,E2 -15041.222} C_VEL
LIN {X 0,Y 324.897,Z 366.343,A -85,B 0,C 180,E1 -15043.256,E2 -15043.256} C_VEL
LIN {X 0,Y 324.92,Z 367.03,A -85,B 0,C 180,E1 -15045.042,E2 -15045.042} C_VEL
LIN {X 0,Y 325.008,Z 366.824,A -85,B 0,C 180,E1 -15046.325,E2 -15046.325} C_VEL
LIN {X 0,Y 325.313,Z 365.748,A -85,B 0,C 180,E1 -15048.101,E2 -15048.101} C_VEL
LIN {X 0,Y 325.847,Z 363.138,A -85,B 0,C 180,E1 -15050.186,E2 -15050.186} C_VEL
LIN {X 0,Y 326.292,Z 360.756,A -85,B 0,C 180,E1 -15051.477,E2 -15051.477} C_VEL
LIN {X 0,Y 327.072,Z 355.811,A -85,B 0,C 180,E1 -15053.421,E2 -15053.421} C_VEL
LIN {X 0,Y 327.774,Z 351.617,A -85,B 0,C 180,E1 -15054.713,E2 -15054.713} C_VEL
LIN {X 0,Y 328.655,Z 346.092,A -85,B 0,C 180,E1 -15056.094,E2 -15056.094} C_VEL
LIN {X 0,Y 329.463,Z 340.258,A -85,B 0,C 180,E1 -15057.297,E2 -15057.297} C_VEL
LIN {X 0,Y 330.579,Z 332.599,A -85,B 0,C 180,E1 -15058.575,E2 -15058.575} C_VEL
LIN {X 0,Y 331.522,Z 325.687,A -85,B 0,C 180,E1 -15059.518,E2 -15059.518} C_VEL
LIN {X 0,Y 332.3,Z 318.33,A -85,B 0,C 180,E1 -15060.355,E2 -15060.355} C_VEL
LIN {X 0,Y 331.681,Z 312.635,A -85,B 0,C 180,E1 -15060.987,E2 -15060.987} C_VEL
LIN {X 0,Y 329.844,Z 303.819,A -85,B 0,C 180,E1 -15061.852,E2 -15061.852} C_VEL
LIN {X 0,Y 327.119,Z 294.044,A -85,B 0,C 180,E1 -15062.662,E2 -15062.662} C_VEL
LIN {X 0,Y 325.647,Z 289.006,A -85,B 0,C 180,E1 -15063.043,E2 -15063.043} C_VEL
LIN {X 0,Y 325.858,Z 285.013,A -85,B 0,C 180,E1 -15067.147,E2 -15067.147} C_VEL
LIN {X 0,Y 326.171,Z 281.354,A -85,B 0,C 180,E1 -15071.054,E2 -15071.054} C_VEL
LIN {X 0,Y 326.336,Z 279.061,A -85,B 0,C 180,E1 -15073.561,E2 -15073.561} C_VEL
LIN {X 0,Y 326.369,Z 276.641,A -85,B 0,C 180,E1 -15076.447,E2 -15076.447} C_VEL
LIN {X 0,Y 326.544,Z 276.624,A -85,B 0,C 180,E1 -15079.788,E2 -15079.788} C_VEL
LIN {X 0,Y 326.613,Z 276.617,A -85,B 0,C 180,E1 -15082.955,E2 -15082.955} C_VEL
LIN {X 0,Y 326.584,Z 276.617,A -85,B 0,C 180,E1 -15086.768,E2 -15086.768} C_VEL
LIN {X 0,Y 326.63,Z 276.613,A -85,B 0,C 180,E1 -15090.341,E2 -15090.341} C_VEL
LIN {X 0,Y 326.632,Z 276.61,A -85,B 0,C 180,E1 -15092.117,E2 -15092.117} C_VEL
LIN {X 0,Y 325.964,Z 276.694,A -85,B 0,C 180,E1 -15093.146,E2 -15093.146} C_VEL
LIN {X 0,Y 323.126,Z 277.048,A -85,B 0,C 180,E1 -15094.821,E2 -15094.821} C_VEL
LIN {X 0,Y 320.712,Z 277.35,A -85,B 0,C 180,E1 -15096.177,E2 -15096.177} C_VEL
LIN {X 0,Y 319.659,Z 277.481,A -85,B 0,C 180,E1 -15097.227,E2 -15097.227} C_VEL
LIN {X 0,Y 319.564,Z 277.492,A -85,B 0,C 180,E1 -15097.583,E2 -15097.583} C_VEL
LIN {X 0,Y 319.673,Z 277.478,A -85,B 0,C 180,E1 -15100.964,E2 -15100.964} C_VEL
LIN {X 0,Y 319.716,Z 277.469,A -85,B 0,C 180,E1 -15105.278,E2 -15105.278} C_VEL
LIN {X 0,Y 319.74,Z 277.465,A -85,B 0,C 180,E1 -15109.875,E2 -15109.875} C_VEL
LIN {X 0,Y 319.896,Z 277.444,A -85,B 0,C 180,E1 -15113.696,E2 -15113.696} C_VEL
LIN {X 0,Y 319.981,Z 277.435,A -85,B 0,C 180,E1 -15117.485,E2 -15117.485} C_VEL
LIN {X 0,Y 320.139,Z 277.42,A -85,B 0,C 180,E1 -15120.002,E2 -15120.002} C_VEL
LIN {X 0,Y 319.979,Z 277.436,A -85,B 0,C 180,E1 -15122.52,E2 -15122.52} C_VEL
LIN {X 0,Y 319.942,Z 277.438,A -85,B 0,C 180,E1 -15126.308,E2 -15126.308} C_VEL
LIN {X 0,Y 319.834,Z 277.458,A -85,B 0,C 180,E1 -15128.85,E2 -15128.85} C_VEL
LIN {X 0,Y 319.675,Z 277.477,A -85,B 0,C 180,E1 -15132.702,E2 -15132.702} C_VEL
LIN {X 0,Y 319.691,Z 277.477,A -85,B 0,C 180,E1 -15135.298,E2 -15135.298} C_VEL
LIN {X 0,Y 319.666,Z 277.479,A -85,B 0,C 180,E1 -15139.258,E2 -15139.258} C_VEL
LIN {X 0,Y 319.549,Z 277.495,A -85,B 0,C 180,E1 -15143.323,E2 -15143.323} C_VEL
LIN {X 0,Y 319.567,Z 277.497,A -85,B 0,C 180,E1 -15146.096,E2 -15146.096} C_VEL
LIN {X 0,Y 319.538,Z 277.5,A -85,B 0,C 180,E1 -15148.941,E2 -15148.941} C_VEL
LIN {X 0,Y 319.519,Z 277.503,A -85,B 0,C 180,E1 -15151.865,E2 -15151.865} C_VEL
LIN {X 0,Y 319.575,Z 277.496,A -85,B 0,C 180,E1 -15155.545,E2 -15155.545} C_VEL
LIN {X 0,Y 319.577,Z 277.492,A -85,B 0,C 180,E1 -15158.009,E2 -15158.009} C_VEL
LIN {X 0,Y 319.566,Z 277.493,A -85,B 0,C 180,E1 -15161.608,E2 -15161.608} C_VEL
LIN {X 0,Y 319.513,Z 277.613,A -85,B 0,C 180,E1 -15165.264,E2 -15165.264} C_VEL
LIN {X 0,Y 320.334,Z 281.843,A -85,B 0,C 180,E1 -15168.841,E2 -15168.841} C_VEL
LIN {X 0,Y 321.086,Z 286.16,A -85,B 0,C 180,E1 -15172.205,E2 -15172.205} C_VEL
LIN {X 0,Y 321.721,Z 290.557,A -85,B 0,C 180,E1 -15175.394,E2 -15175.394} C_VEL
LIN {X 0,Y 321.593,Z 293.884,A -85,B 0,C 180,E1 -15177.63,E2 -15177.63} C_VEL
LIN {X 0,Y 320.629,Z 299.583,A -85,B 0,C 180,E1 -15181.258,E2 -15181.258} C_VEL
LIN {X 0,Y 319.669,Z 306.208,A -85,B 0,C 180,E1 -15185.311,E2 -15185.311} C_VEL
LIN {X 0,Y 318.891,Z 312.999,A -85,B 0,C 180,E1 -15189.354,E2 -15189.354} C_VEL
LIN {X 0,Y 318.791,Z 315.103,A -85,B 0,C 180,E1 -15190.466,E2 -15190.466} C_VEL
LIN {X 0,Y 321.378,Z 327.463,A -85,B 0,C 180,E1 -15191.296,E2 -15191.296} C_VEL
LIN {X 0,Y 322.691,Z 336.744,A -85,B 0,C 180,E1 -15192.081,E2 -15192.081} C_VEL
LIN {X 0,Y 323.441,Z 345.388,A -85,B 0,C 180,E1 -15192.957,E2 -15192.957} C_VEL
LIN {X 0,Y 323.504,Z 353.499,A -85,B 0,C 180,E1 -15193.921,E2 -15193.921} C_VEL
LIN {X 0,Y 322.606,Z 361.38,A -85,B 0,C 180,E1 -15195.009,E2 -15195.009} C_VEL
LIN {X 0,Y 321.504,Z 367.925,A -85,B 0,C 180,E1 -15196.088,E2 -15196.088} C_VEL
LIN {X 0,Y 320.54,Z 374.161,A -85,B 0,C 180,E1 -15197.337,E2 -15197.337} C_VEL
LIN {X 0,Y 319.764,Z 379.358,A -85,B 0,C 180,E1 -15198.593,E2 -15198.593} C_VEL
LIN {X 0,Y 319.104,Z 383.708,A -85,B 0,C 180,E1 -15199.854,E2 -15199.854} C_VEL
LIN {X 0,Y 318.393,Z 388.87,A -85,B 0,C 180,E1 -15201.753,E2 -15201.753} C_VEL
LIN {X 0,Y 317.985,Z 392.678,A -85,B 0,C 180,E1 -15203.657,E2 -15203.657} C_VEL
LIN {X 0,Y 317.871,Z 394.437,A -85,B 0,C 180,E1 -15204.928,E2 -15204.928} C_VEL
LIN {X 0,Y 317.872,Z 395.71,A -85,B 0,C 180,E1 -15206.199,E2 -15206.199} C_VEL
LIN {X 0,Y 317.823,Z 396.511,A -85,B 0,C 180,E1 -15207.467,E2 -15207.467} C_VEL
LIN {X 0,Y 317.868,Z 396.834,A -85,B 0,C 180,E1 -15208.735,E2 -15208.735} C_VEL
LIN {X 0,Y 317.951,Z 396.562,A -85,B 0,C 180,E1 -15210.002,E2 -15210.002} C_VEL
LIN {X 0,Y 317.917,Z 395.793,A -85,B 0,C 180,E1 -15211.268,E2 -15211.268} C_VEL
LIN {X 0,Y 317.862,Z 394.541,A -85,B 0,C 180,E1 -15212.536,E2 -15212.536} C_VEL
LIN {X 0,Y 317.95,Z 391.632,A -85,B 0,C 180,E1 -15214.439,E2 -15214.439} C_VEL
LIN {X 0,Y 317.954,Z 388.485,A -85,B 0,C 180,E1 -15215.906,E2 -15215.906} C_VEL
LIN {X 0,Y 318.286,Z 382.758,A -85,B 0,C 180,E1 -15217.934,E2 -15217.934} C_VEL
LIN {X 0,Y 318.642,Z 376.799,A -85,B 0,C 180,E1 -15219.523,E2 -15219.523} C_VEL
LIN {X 0,Y 319.245,Z 369.23,A -85,B 0,C 180,E1 -15221.108,E2 -15221.108} C_VEL
LIN {X 0,Y 319.746,Z 362.78,A -85,B 0,C 180,E1 -15222.215,E2 -15222.215} C_VEL
LIN {X 0,Y 320.354,Z 356.218,A -85,B 0,C 180,E1 -15223.158,E2 -15223.158} C_VEL
LIN {X 0,Y 320.834,Z 349.767,A -85,B 0,C 180,E1 -15223.945,E2 -15223.945} C_VEL
LIN {X 0,Y 320.39,Z 341.564,A -85,B 0,C 180,E1 -15224.79,E2 -15224.79} C_VEL
LIN {X 0,Y 319.744,Z 332.447,A -85,B 0,C 180,E1 -15225.54,E2 -15225.54} C_VEL
LIN {X 0,Y 318.897,Z 322.579,A -85,B 0,C 180,E1 -15226.156,E2 -15226.156} C_VEL
LIN {X 0,Y 318.189,Z 315.49,A -85,B 0,C 180,E1 -15226.523,E2 -15226.523} C_VEL
LIN {X 0,Y 318.522,Z 309.311,A -85,B 0,C 180,E1 -15230,E2 -15230} C_VEL
LIN {X 0,Y 319.022,Z 303.351,A -85,B 0,C 180,E1 -15233.363,E2 -15233.363} C_VEL
LIN {X 0,Y 319.605,Z 297.417,A -85,B 0,C 180,E1 -15236.796,E2 -15236.796} C_VEL
LIN {X 0,Y 320.352,Z 291.428,A -85,B 0,C 180,E1 -15240.305,E2 -15240.305} C_VEL
LIN {X 0,Y 320.928,Z 286.631,A -85,B 0,C 180,E1 -15243.196,E2 -15243.196} C_VEL
LIN {X 0,Y 320.556,Z 282.563,A -85,B 0,C 180,E1 -15245.784,E2 -15245.784} C_VEL
LIN {X 0,Y 319.648,Z 277.48,A -85,B 0,C 180,E1 -15249.208,E2 -15249.208} C_VEL
LIN {X 0,Y 319.532,Z 277.494,A -85,B 0,C 180,E1 -15253.46,E2 -15253.46} C_VEL
LIN {X 0,Y 319.564,Z 277.488,A -85,B 0,C 180,E1 -15257.016,E2 -15257.016} C_VEL
LIN {X 0,Y 319.557,Z 277.49,A -85,B 0,C 180,E1 -15260.37,E2 -15260.37} C_VEL
LIN {X 0,Y 319.568,Z 277.492,A -85,B 0,C 180,E1 -15263.572,E2 -15263.572} C_VEL
LIN {X 0,Y 319.588,Z 277.485,A -85,B 0,C 180,E1 -15266.686,E2 -15266.686} C_VEL
LIN {X 0,Y 319.602,Z 277.488,A -85,B 0,C 180,E1 -15269.616,E2 -15269.616} C_VEL
LIN {X 0,Y 319.619,Z 277.481,A -85,B 0,C 180,E1 -15272.497,E2 -15272.497} C_VEL
LIN {X 0,Y 319.614,Z 277.487,A -85,B 0,C 180,E1 -15275.303,E2 -15275.303} C_VEL
LIN {X 0,Y 319.592,Z 277.489,A -85,B 0,C 180,E1 -15279.398,E2 -15279.398} C_VEL
LIN {X 0,Y 319.66,Z 277.479,A -85,B 0,C 180,E1 -15283.39,E2 -15283.39} C_VEL
LIN {X 0,Y 319.741,Z 277.466,A -85,B 0,C 180,E1 -15286.006,E2 -15286.006} C_VEL
LIN {X 0,Y 319.744,Z 277.466,A -85,B 0,C 180,E1 -15289.87,E2 -15289.87} C_VEL
LIN {X 0,Y 319.943,Z 277.441,A -85,B 0,C 180,E1 -15293.692,E2 -15293.692} C_VEL
LIN {X 0,Y 319.996,Z 277.434,A -85,B 0,C 180,E1 -15297.48,E2 -15297.48} C_VEL
LIN {X 0,Y 320.138,Z 277.417,A -85,B 0,C 180,E1 -15299.998,E2 -15299.998} C_VEL
LIN {X 0,Y 319.997,Z 277.44,A -85,B 0,C 180,E1 -15302.515,E2 -15302.515} C_VEL
LIN {X 0,Y 319.937,Z 277.443,A -85,B 0,C 180,E1 -15306.625,E2 -15306.625} C_VEL
LIN {X 0,Y 319.762,Z 277.467,A -85,B 0,C 180,E1 -15310.124,E2 -15310.124} C_VEL
LIN {X 0,Y 319.734,Z 277.468,A -85,B 0,C 180,E1 -15314.721,E2 -15314.721} C_VEL
LIN {X 0,Y 319.691,Z 277.472,A -85,B 0,C 180,E1 -15319.035,E2 -15319.035} C_VEL
LIN {X 0,Y 319.571,Z 277.488,A -85,B 0,C 180,E1 -15323.316,E2 -15323.316} C_VEL
LIN {X 0,Y 319.633,Z 277.483,A -85,B 0,C 180,E1 -15326.085,E2 -15326.085} C_VEL
LIN {X 0,Y 319.578,Z 277.487,A -85,B 0,C 180,E1 -15328.931,E2 -15328.931} C_VEL
LIN {X 0,Y 319.528,Z 277.497,A -85,B 0,C 180,E1 -15331.859,E2 -15331.859} C_VEL
LIN {X 0,Y 319.577,Z 277.492,A -85,B 0,C 180,E1 -15335.54,E2 -15335.54} C_VEL
LIN {X 0,Y 319.596,Z 277.486,A -85,B 0,C 180,E1 -15338.001,E2 -15338.001} C_VEL
LIN {X 0,Y 319.596,Z 277.488,A -85,B 0,C 180,E1 -15341.609,E2 -15341.609} C_VEL
LIN {X 0,Y 319.638,Z 277.484,A -85,B 0,C 180,E1 -15345.282,E2 -15345.282} C_VEL
LIN {X 0,Y 319.574,Z 277.489,A -85,B 0,C 180,E1 -15348.717,E2 -15348.717} C_VEL
LIN {X 0,Y 319.573,Z 277.488,A -85,B 0,C 180,E1 -15352.34,E2 -15352.34} C_VEL
LIN {X 0,Y 319.55,Z 277.494,A -85,B 0,C 180,E1 -15355.12,E2 -15355.12} C_VEL
LIN {X 0,Y 319.559,Z 277.493,A -85,B 0,C 180,E1 -15359.055,E2 -15359.055} C_VEL
LIN {X 0,Y 319.597,Z 277.487,A -85,B 0,C 180,E1 -15362.495,E2 -15362.495} C_VEL
LIN {X 0,Y 319.596,Z 277.485,A -85,B 0,C 180,E1 -15365.302,E2 -15365.302} C_VEL
LIN {X 0,Y 319.584,Z 277.487,A -85,B 0,C 180,E1 -15368.045,E2 -15368.045} C_VEL
LIN {X 0,Y 319.523,Z 277.494,A -85,B 0,C 180,E1 -15371.039,E2 -15371.039} C_VEL
LIN {X 0,Y 319.162,Z 277.541,A -85,B 0,C 180,E1 -15374.677,E2 -15374.677} C_VEL
LIN {X 0,Y 319.039,Z 277.556,A -85,B 0,C 180,E1 -15375.975,E2 -15375.975} C_VEL
LIN {X 0,Y 318.858,Z 277.945,A -85,B 0,C 180,E1 -15377.265,E2 -15377.265} C_VEL
LIN {X 0,Y 318.697,Z 281.838,A -85,B 0,C 180,E1 -15381.118,E2 -15381.118} C_VEL
LIN {X 0,Y 318.713,Z 284.455,A -85,B 0,C 180,E1 -15383.668,E2 -15383.668} C_VEL
LIN {X 0,Y 318.657,Z 287.085,A -85,B 0,C 180,E1 -15386.205,E2 -15386.205} C_VEL
LIN {X 0,Y 318.502,Z 288.772,A -85,B 0,C 180,E1 -15387.667,E2 -15387.667} C_VEL
LIN {X 0,Y 320.206,Z 299.18,A -85,B 0,C 180,E1 -15388.269,E2 -15388.269} C_VEL
LIN {X 0,Y 321.381,Z 307.523,A -85,B 0,C 180,E1 -15388.902,E2 -15388.902} C_VEL
LIN {X 0,Y 322.018,Z 312.734,A -85,B 0,C 180,E1 -15389.373,E2 -15389.373} C_VEL
LIN {X 0,Y 321.258,Z 323.219,A -85,B 0,C 180,E1 -15390.468,E2 -15390.468} C_VEL
LIN {X 0,Y 320.635,Z 331.396,A -85,B 0,C 180,E1 -15391.568,E2 -15391.568} C_VEL
LIN {X 0,Y 319.97,Z 339.01,A -85,B 0,C 180,E1 -15392.831,E2 -15392.831} C_VEL
LIN {X 0,Y 319.454,Z 345.26,A -85,B 0,C 180,E1 -15394.098,E2 -15394.098} C_VEL
LIN {X 0,Y 319.003,Z 350.457,A -85,B 0,C 180,E1 -15395.371,E2 -15395.371} C_VEL
LIN {X 0,Y 318.677,Z 355.046,A -85,B 0,C 180,E1 -15396.735,E2 -15396.735} C_VEL
LIN {X 0,Y 318.327,Z 359.145,A -85,B 0,C 180,E1 -15398.249,E2 -15398.249} C_VEL
LIN {X 0,Y 318.098,Z 361.907,A -85,B 0,C 180,E1 -15399.536,E2 -15399.536} C_VEL
LIN {X 0,Y 317.859,Z 364.927,A -85,B 0,C 180,E1 -15401.476,E2 -15401.476} C_VEL
LIN {X 0,Y 317.825,Z 366.707,A -85,B 0,C 180,E1 -15403.369,E2 -15403.369} C_VEL
LIN {X 0,Y 317.841,Z 367.391,A -85,B 0,C 180,E1 -15405.385,E2 -15405.385} C_VEL
LIN {X 0,Y 317.993,Z 367.101,A -85,B 0,C 180,E1 -15406.695,E2 -15406.695} C_VEL
LIN {X 0,Y 318.267,Z 366.072,A -85,B 0,C 180,E1 -15408.292,E2 -15408.292} C_VEL
LIN {X 0,Y 318.898,Z 363.053,A -85,B 0,C 180,E1 -15410.645,E2 -15410.645} C_VEL
LIN {X 0,Y 319.614,Z 359.169,A -85,B 0,C 180,E1 -15412.56,E2 -15412.56} C_VEL
LIN {X 0,Y 320.266,Z 355.451,A -85,B 0,C 180,E1 -15413.95,E2 -15413.95} C_VEL
LIN {X 0,Y 321.067,Z 351.103,A -85,B 0,C 180,E1 -15415.266,E2 -15415.266} C_VEL
LIN {X 0,Y 321.999,Z 345.221,A -85,B 0,C 180,E1 -15416.717,E2 -15416.717} C_VEL
LIN {X 0,Y 322.872,Z 339.361,A -85,B 0,C 180,E1 -15417.902,E2 -15417.902} C_VEL
LIN {X 0,Y 323.899,Z 332.523,A -85,B 0,C 180,E1 -15419.043,E2 -15419.043} C_VEL
LIN {X 0,Y 325.076,Z 324.362,A -85,B 0,C 180,E1 -15420.149,E2 -15420.149} C_VEL
LIN {X 0,Y 325.567,Z 318.025,A -85,B 0,C 180,E1 -15420.871,E2 -15420.871} C_VEL
LIN {X 0,Y 324.246,Z 310.081,A -85,B 0,C 180,E1 -15421.76,E2 -15421.76} C_VEL
LIN {X 0,Y 322.176,Z 301.538,A -85,B 0,C 180,E1 -15422.593,E2 -15422.593} C_VEL
LIN {X 0,Y 319.4,Z 292.043,A -85,B 0,C 180,E1 -15423.371,E2 -15423.371} C_VEL
LIN {X 0,Y 318.633,Z 289.342,A -85,B 0,C 180,E1 -15423.604,E2 -15423.604} C_VEL
LIN {X 0,Y 318.883,Z 285.068,A -85,B 0,C 180,E1 -15428.103,E2 -15428.103} C_VEL
LIN {X 0,Y 319.151,Z 281.919,A -85,B 0,C 180,E1 -15431.526,E2 -15431.526} C_VEL
LIN {X 0,Y 319.363,Z 279.056,A -85,B 0,C 180,E1 -15434.762,E2 -15434.762} C_VEL
LIN {X 0,Y 319.348,Z 277.525,A -85,B 0,C 180,E1 -15436.569,E2 -15436.569} C_VEL
LIN {X 0,Y 319.525,Z 277.496,A -85,B 0,C 180,E1 -15440.372,E2 -15440.372} C_VEL
LIN {X 0,Y 319.541,Z 277.497,A -85,B 0,C 180,E1 -15443.574,E2 -15443.574} C_VEL
LIN {X 0,Y 319.559,Z 277.493,A -85,B 0,C 180,E1 -15446.688,E2 -15446.688} C_VEL
LIN {X 0,Y 319.566,Z 277.492,A -85,B 0,C 180,E1 -15449.617,E2 -15449.617} C_VEL
LIN {X 0,Y 319.588,Z 277.49,A -85,B 0,C 180,E1 -15452.499,E2 -15452.499} C_VEL
LIN {X 0,Y 319.587,Z 277.49,A -85,B 0,C 180,E1 -15455.306,E2 -15455.306} C_VEL
LIN {X 0,Y 319.564,Z 277.492,A -85,B 0,C 180,E1 -15457.583,E2 -15457.583} C_VEL
LIN {X 0,Y 318.883,Z 277.577,A -85,B 0,C 180,E1 -15458.636,E2 -15458.636} C_VEL
LIN {X 0,Y 316.07,Z 277.928,A -85,B 0,C 180,E1 -15460.351,E2 -15460.351} C_VEL
LIN {X 0,Y 313.696,Z 278.223,A -85,B 0,C 180,E1 -15461.741,E2 -15461.741} C_VEL
LIN {X 0,Y 312.673,Z 278.347,A -85,B 0,C 180,E1 -15462.816,E2 -15462.816} C_VEL
LIN {X 0,Y 312.586,Z 278.357,A -85,B 0,C 180,E1 -15463.18,E2 -15463.18} C_VEL
LIN {X 0,Y 312.68,Z 278.344,A -85,B 0,C 180,E1 -15465.688,E2 -15465.688} C_VEL
LIN {X 0,Y 312.686,Z 278.344,A -85,B 0,C 180,E1 -15469.644,E2 -15469.644} C_VEL
LIN {X 0,Y 312.804,Z 278.334,A -85,B 0,C 180,E1 -15472.255,E2 -15472.255} C_VEL
LIN {X 0,Y 312.696,Z 278.347,A -85,B 0,C 180,E1 -15474.844,E2 -15474.844} C_VEL
LIN {X 0,Y 312.982,Z 278.307,A -85,B 0,C 180,E1 -15478.716,E2 -15478.716} C_VEL
LIN {X 0,Y 312.979,Z 278.308,A -85,B 0,C 180,E1 -15481.289,E2 -15481.289} C_VEL
LIN {X 0,Y 312.708,Z 278.345,A -85,B 0,C 180,E1 -15485.16,E2 -15485.16} C_VEL
LIN {X 0,Y 312.862,Z 278.326,A -85,B 0,C 180,E1 -15487.748,E2 -15487.748} C_VEL
LIN {X 0,Y 312.662,Z 278.352,A -85,B 0,C 180,E1 -15491.674,E2 -15491.674} C_VEL
LIN {X 0,Y 312.692,Z 278.348,A -85,B 0,C 180,E1 -15494.89,E2 -15494.89} C_VEL
LIN {X 0,Y 312.622,Z 278.356,A -85,B 0,C 180,E1 -15499.238,E2 -15499.238} C_VEL
LIN {X 0,Y 312.517,Z 278.372,A -85,B 0,C 180,E1 -15502.782,E2 -15502.782} C_VEL
LIN {X 0,Y 312.527,Z 278.372,A -85,B 0,C 180,E1 -15505.912,E2 -15505.912} C_VEL
LIN {X 0,Y 312.491,Z 278.377,A -85,B 0,C 180,E1 -15509.658,E2 -15509.658} C_VEL
LIN {X 0,Y 312.515,Z 278.377,A -85,B 0,C 180,E1 -15513.691,E2 -15513.691} C_VEL
LIN {X 0,Y 312.536,Z 278.371,A -85,B 0,C 180,E1 -15517.386,E2 -15517.386} C_VEL
LIN {X 0,Y 312.497,Z 278.373,A -85,B 0,C 180,E1 -15520.71,E2 -15520.71} C_VEL
LIN {X 0,Y 312.462,Z 278.38,A -85,B 0,C 180,E1 -15524.21,E2 -15524.21} C_VEL
LIN {X 0,Y 312.45,Z 278.406,A -85,B 0,C 180,E1 -15524.626,E2 -15524.626} C_VEL
LIN {X 0,Y 313.355,Z 282.974,A -85,B 0,C 180,E1 -15528.63,E2 -15528.63} C_VEL
LIN {X 0,Y 314.279,Z 288.321,A -85,B 0,C 180,E1 -15532.861,E2 -15532.861} C_VEL
LIN {X 0,Y 314.731,Z 292.696,A -85,B 0,C 180,E1 -15536.067,E2 -15536.067} C_VEL
LIN {X 0,Y 314.415,Z 295.775,A -85,B 0,C 180,E1 -15538.149,E2 -15538.149} C_VEL
LIN {X 0,Y 313.414,Z 301.582,A -85,B 0,C 180,E1 -15541.909,E2 -15541.909} C_VEL
LIN {X 0,Y 312.579,Z 307.204,A -85,B 0,C 180,E1 -15545.423,E2 -15545.423} C_VEL
LIN {X 0,Y 311.742,Z 314.462,A -85,B 0,C 180,E1 -15549.85,E2 -15549.85} C_VEL
LIN {X 0,Y 314.471,Z 327.336,A -85,B 0,C 180,E1 -15550.778,E2 -15550.778} C_VEL
LIN {X 0,Y 315.78,Z 336.01,A -85,B 0,C 180,E1 -15551.535,E2 -15551.535} C_VEL
LIN {X 0,Y 316.583,Z 345.243,A -85,B 0,C 180,E1 -15552.496,E2 -15552.496} C_VEL
LIN {X 0,Y 316.757,Z 352.68,A -85,B 0,C 180,E1 -15553.403,E2 -15553.403} C_VEL
LIN {X 0,Y 316.081,Z 359.619,A -85,B 0,C 180,E1 -15554.362,E2 -15554.362} C_VEL
LIN {X 0,Y 314.964,Z 366.396,A -85,B 0,C 180,E1 -15555.463,E2 -15555.463} C_VEL
LIN {X 0,Y 313.883,Z 372.831,A -85,B 0,C 180,E1 -15556.734,E2 -15556.734} C_VEL
LIN {X 0,Y 312.998,Z 378.199,A -85,B 0,C 180,E1 -15558.014,E2 -15558.014} C_VEL
LIN {X 0,Y 312.091,Z 383.656,A -85,B 0,C 180,E1 -15559.623,E2 -15559.623} C_VEL
LIN {X 0,Y 311.34,Z 388.757,A -85,B 0,C 180,E1 -15561.564,E2 -15561.564} C_VEL
LIN {X 0,Y 310.917,Z 392.505,A -85,B 0,C 180,E1 -15563.512,E2 -15563.512} C_VEL
LIN {X 0,Y 310.788,Z 394.219,A -85,B 0,C 180,E1 -15564.812,E2 -15564.812} C_VEL
LIN {X 0,Y 310.78,Z 395.446,A -85,B 0,C 180,E1 -15566.112,E2 -15566.112} C_VEL
LIN {X 0,Y 310.744,Z 396.203,A -85,B 0,C 180,E1 -15567.409,E2 -15567.409} C_VEL
LIN {X 0,Y 310.775,Z 396.497,A -85,B 0,C 180,E1 -15568.706,E2 -15568.706} C_VEL
LIN {X 0,Y 310.859,Z 396.209,A -85,B 0,C 180,E1 -15570.002,E2 -15570.002} C_VEL
LIN {X 0,Y 310.822,Z 395.395,A -85,B 0,C 180,E1 -15571.297,E2 -15571.297} C_VEL
LIN {X 0,Y 310.783,Z 394.098,A -85,B 0,C 180,E1 -15572.594,E2 -15572.594} C_VEL
LIN {X 0,Y 310.86,Z 391.14,A -85,B 0,C 180,E1 -15574.54,E2 -15574.54} C_VEL
LIN {X 0,Y 310.939,Z 386.882,A -85,B 0,C 180,E1 -15576.491,E2 -15576.491} C_VEL
LIN {X 0,Y 311.281,Z 380.986,A -85,B 0,C 180,E1 -15578.441,E2 -15578.441} C_VEL
LIN {X 0,Y 311.582,Z 376.066,A -85,B 0,C 180,E1 -15579.741,E2 -15579.741} C_VEL
LIN {X 0,Y 312.096,Z 370.137,A -85,B 0,C 180,E1 -15581.037,E2 -15581.037} C_VEL
LIN {X 0,Y 312.694,Z 362.902,A -85,B 0,C 180,E1 -15582.33,E2 -15582.33} C_VEL
LIN {X 0,Y 313.453,Z 355.195,A -85,B 0,C 180,E1 -15583.453,E2 -15583.453} C_VEL
LIN {X 0,Y 313.723,Z 348.547,A -85,B 0,C 180,E1 -15584.267,E2 -15584.267} C_VEL
LIN {X 0,Y 313.272,Z 340.105,A -85,B 0,C 180,E1 -15585.134,E2 -15585.134} C_VEL
LIN {X 0,Y 312.608,Z 330.631,A -85,B 0,C 180,E1 -15585.904,E2 -15585.904} C_VEL
LIN {X 0,Y 311.71,Z 320.583,A -85,B 0,C 180,E1 -15586.519,E2 -15586.519} C_VEL
LIN {X 0,Y 311.143,Z 315.159,A -85,B 0,C 180,E1 -15586.824,E2 -15586.824} C_VEL
LIN {X 0,Y 311.619,Z 307.652,A -85,B 0,C 180,E1 -15591.154,E2 -15591.154} C_VEL
LIN {X 0,Y 312.258,Z 300.558,A -85,B 0,C 180,E1 -15595.319,E2 -15595.319} C_VEL
LIN {X 0,Y 312.943,Z 294.621,A -85,B 0,C 180,E1 -15598.851,E2 -15598.851} C_VEL
LIN {X 0,Y 313.848,Z 288.62,A -85,B 0,C 180,E1 -15602.511,E2 -15602.511} C_VEL
LIN {X 0,Y 313.773,Z 284.994,A -85,B 0,C 180,E1 -15604.832,E2 -15604.832} C_VEL
LIN {X 0,Y 312.86,Z 280.075,A -85,B 0,C 180,E1 -15608.163,E2 -15608.163} C_VEL
LIN {X 0,Y 312.574,Z 278.362,A -85,B 0,C 180,E1 -15609.422,E2 -15609.422} C_VEL
LIN {X 0,Y 312.5,Z 278.37,A -85,B 0,C 180,E1 -15612.432,E2 -15612.432} C_VEL
LIN {X 0,Y 312.468,Z 278.376,A -85,B 0,C 180,E1 -15616.035,E2 -15616.035} C_VEL
LIN {X 0,Y 312.515,Z 278.371,A -85,B 0,C 180,E1 -15619.874,E2 -15619.874} C_VEL
LIN {X 0,Y 312.545,Z 278.365,A -85,B 0,C 180,E1 -15624.05,E2 -15624.05} C_VEL
LIN {X 0,Y 312.515,Z 278.37,A -85,B 0,C 180,E1 -15627.333,E2 -15627.333} C_VEL
LIN {X 0,Y 312.563,Z 278.364,A -85,B 0,C 180,E1 -15631.275,E2 -15631.275} C_VEL
LIN {X 0,Y 312.595,Z 278.357,A -85,B 0,C 180,E1 -15634.71,E2 -15634.71} C_VEL
LIN {X 0,Y 312.574,Z 278.361,A -85,B 0,C 180,E1 -15637.526,E2 -15637.526} C_VEL
LIN {X 0,Y 312.576,Z 278.36,A -85,B 0,C 180,E1 -15641.651,E2 -15641.651} C_VEL
LIN {X 0,Y 312.695,Z 278.344,A -85,B 0,C 180,E1 -15645.684,E2 -15645.684} C_VEL
LIN {X 0,Y 312.694,Z 278.344,A -85,B 0,C 180,E1 -15649.639,E2 -15649.639} C_VEL
LIN {X 0,Y 312.899,Z 278.319,A -85,B 0,C 180,E1 -15653.55,E2 -15653.55} C_VEL
LIN {X 0,Y 312.942,Z 278.313,A -85,B 0,C 180,E1 -15657.423,E2 -15657.423} C_VEL
LIN {X 0,Y 313.091,Z 278.295,A -85,B 0,C 180,E1 -15659.998,E2 -15659.998} C_VEL
LIN {X 0,Y 312.944,Z 278.318,A -85,B 0,C 180,E1 -15662.572,E2 -15662.572} C_VEL
LIN {X 0,Y 312.902,Z 278.322,A -85,B 0,C 180,E1 -15666.607,E2 -15666.607} C_VEL
LIN {X 0,Y 312.792,Z 278.332,A -85,B 0,C 180,E1 -15669.047,E2 -15669.047} C_VEL
LIN {X 0,Y 312.638,Z 278.351,A -85,B 0,C 180,E1 -15672.988,E2 -15672.988} C_VEL
LIN {X 0,Y 312.641,Z 278.352,A -85,B 0,C 180,E1 -15675.647,E2 -15675.647} C_VEL
LIN {X 0,Y 312.632,Z 278.352,A -85,B 0,C 180,E1 -15679.233,E2 -15679.233} C_VEL
LIN {X 0,Y 312.546,Z 278.362,A -85,B 0,C 180,E1 -15682.786,E2 -15682.786} C_VEL
LIN {X 0,Y 312.602,Z 278.36,A -85,B 0,C 180,E1 -15685.932,E2 -15685.932} C_VEL
LIN {X 0,Y 312.536,Z 278.368,A -85,B 0,C 180,E1 -15689.648,E2 -15689.648} C_VEL
LIN {X 0,Y 312.516,Z 278.371,A -85,B 0,C 180,E1 -15693.686,E2 -15693.686} C_VEL
LIN {X 0,Y 312.549,Z 278.366,A -85,B 0,C 180,E1 -15697.378,E2 -15697.378} C_VEL
LIN {X 0,Y 312.53,Z 278.365,A -85,B 0,C 180,E1 -15700.699,E2 -15700.699} C_VEL
LIN {X 0,Y 312.588,Z 278.357,A -85,B 0,C 180,E1 -15704.181,E2 -15704.181} C_VEL
LIN {X 0,Y 312.548,Z 278.363,A -85,B 0,C 180,E1 -15707.901,E2 -15707.901} C_VEL
LIN {X 0,Y 312.535,Z 278.364,A -85,B 0,C 180,E1 -15711.905,E2 -15711.905} C_VEL
LIN {X 0,Y 312.496,Z 278.369,A -85,B 0,C 180,E1 -15715.787,E2 -15715.787} C_VEL
LIN {X 0,Y 312.512,Z 278.372,A -85,B 0,C 180,E1 -15718.851,E2 -15718.851} C_VEL
LIN {X 0,Y 312.562,Z 278.36,A -85,B 0,C 180,E1 -15721.822,E2 -15721.822} C_VEL
LIN {X 0,Y 312.575,Z 278.364,A -85,B 0,C 180,E1 -15724.708,E2 -15724.708} C_VEL
LIN {X 0,Y 312.575,Z 278.359,A -85,B 0,C 180,E1 -15727.526,E2 -15727.526} C_VEL
LIN {X 0,Y 312.485,Z 278.372,A -85,B 0,C 180,E1 -15730.83,E2 -15730.83} C_VEL
LIN {X 0,Y 312.141,Z 278.418,A -85,B 0,C 180,E1 -15734.323,E2 -15734.323} C_VEL
LIN {X 0,Y 311.835,Z 278.456,A -85,B 0,C 180,E1 -15736.973,E2 -15736.973} C_VEL
LIN {X 0,Y 311.631,Z 282.318,A -85,B 0,C 180,E1 -15740.915,E2 -15740.915} C_VEL
LIN {X 0,Y 311.673,Z 284.969,A -85,B 0,C 180,E1 -15743.525,E2 -15743.525} C_VEL
LIN {X 0,Y 311.477,Z 288.67,A -85,B 0,C 180,E1 -15747.088,E2 -15747.088} C_VEL
LIN {X 0,Y 311.463,Z 288.966,A -85,B 0,C 180,E1 -15747.371,E2 -15747.371} C_VEL
LIN {X 0,Y 313.305,Z 300.377,A -85,B 0,C 180,E1 -15748.07,E2 -15748.07} C_VEL
LIN {X 0,Y 314.434,Z 308.539,A -85,B 0,C 180,E1 -15748.718,E2 -15748.718} C_VEL
LIN {X 0,Y 315.027,Z 313.765,A -85,B 0,C 180,E1 -15749.199,E2 -15749.199} C_VEL
LIN {X 0,Y 314.245,Z 324.019,A -85,B 0,C 180,E1 -15750.319,E2 -15750.319} C_VEL
LIN {X 0,Y 313.588,Z 332.122,A -85,B 0,C 180,E1 -15751.443,E2 -15751.443} C_VEL
LIN {X 0,Y 312.978,Z 338.818,A -85,B 0,C 180,E1 -15752.572,E2 -15752.572} C_VEL
LIN {X 0,Y 312.472,Z 345.149,A -85,B 0,C 180,E1 -15753.867,E2 -15753.867} C_VEL
LIN {X 0,Y 311.955,Z 350.428,A -85,B 0,C 180,E1 -15755.169,E2 -15755.169} C_VEL
LIN {X 0,Y 311.679,Z 354.81,A -85,B 0,C 180,E1 -15756.472,E2 -15756.472} C_VEL
LIN {X 0,Y 311.339,Z 358.469,A -85,B 0,C 180,E1 -15757.782,E2 -15757.782} C_VEL
LIN {X 0,Y 311.091,Z 361.47,A -85,B 0,C 180,E1 -15759.097,E2 -15759.097} C_VEL
LIN {X 0,Y 310.854,Z 363.824,A -85,B 0,C 180,E1 -15760.419,E2 -15760.419} C_VEL
LIN {X 0,Y 310.77,Z 365.547,A -85,B 0,C 180,E1 -15761.742,E2 -15761.742} C_VEL
LIN {X 0,Y 310.739,Z 367.059,A -85,B 0,C 180,E1 -15763.475,E2 -15763.475} C_VEL
LIN {X 0,Y 310.8,Z 367.687,A -85,B 0,C 180,E1 -15765.743,E2 -15765.743} C_VEL
LIN {X 0,Y 310.962,Z 367.369,A -85,B 0,C 180,E1 -15767.084,E2 -15767.084} C_VEL
LIN {X 0,Y 311.234,Z 366.397,A -85,B 0,C 180,E1 -15768.496,E2 -15768.496} C_VEL
LIN {X 0,Y 311.754,Z 364.136,A -85,B 0,C 180,E1 -15770.45,E2 -15770.45} C_VEL
LIN {X 0,Y 312.499,Z 360.364,A -85,B 0,C 180,E1 -15772.476,E2 -15772.476} C_VEL
LIN {X 0,Y 313.501,Z 355.103,A -85,B 0,C 180,E1 -15774.5,E2 -15774.5} C_VEL
LIN {X 0,Y 314.578,Z 349.383,A -85,B 0,C 180,E1 -15776.181,E2 -15776.181} C_VEL
LIN {X 0,Y 315.775,Z 342.015,A -85,B 0,C 180,E1 -15777.862,E2 -15777.862} C_VEL
LIN {X 0,Y 316.984,Z 334.581,A -85,B 0,C 180,E1 -15779.192,E2 -15779.192} C_VEL
LIN {X 0,Y 317.994,Z 327.867,A -85,B 0,C 180,E1 -15780.183,E2 -15780.183} C_VEL
LIN {X 0,Y 318.912,Z 320.26,A -85,B 0,C 180,E1 -15781.114,E2 -15781.114} C_VEL
LIN {X 0,Y 317.706,Z 312.265,A -85,B 0,C 180,E1 -15782.064,E2 -15782.064} C_VEL
LIN {X 0,Y 315.518,Z 302.849,A -85,B 0,C 180,E1 -15783.033,E2 -15783.033} C_VEL
LIN {X 0,Y 312.776,Z 293.74,A -85,B 0,C 180,E1 -15783.833,E2 -15783.833} C_VEL
LIN {X 0,Y 311.602,Z 289.701,A -85,B 0,C 180,E1 -15784.151,E2 -15784.151} C_VEL
LIN {X 0,Y 311.842,Z 286.178,A -85,B 0,C 180,E1 -15787.932,E2 -15787.932} C_VEL
LIN {X 0,Y 312.172,Z 282.528,A -85,B 0,C 180,E1 -15792.023,E2 -15792.023} C_VEL
LIN {X 0,Y 312.306,Z 280.592,A -85,B 0,C 180,E1 -15794.233,E2 -15794.233} C_VEL
LIN {X 0,Y 312.344,Z 279.057,A -85,B 0,C 180,E1 -15796.054,E2 -15796.054} C_VEL
LIN {X 0,Y 312.364,Z 278.389,A -85,B 0,C 180,E1 -15797.94,E2 -15797.94} C_VEL
LIN {X 0,Y 312.516,Z 278.372,A -85,B 0,C 180,E1 -15801.912,E2 -15801.912} C_VEL
LIN {X 0,Y 312.488,Z 278.375,A -85,B 0,C 180,E1 -15805.791,E2 -15805.791} C_VEL
LIN {X 0,Y 312.502,Z 278.372,A -85,B 0,C 180,E1 -15808.855,E2 -15808.855} C_VEL
LIN {X 0,Y 312.552,Z 278.364,A -85,B 0,C 180,E1 -15811.826,E2 -15811.826} C_VEL
LIN {X 0,Y 312.568,Z 278.363,A -85,B 0,C 180,E1 -15814.713,E2 -15814.713} C_VEL
LIN {X 0,Y 312.523,Z 278.365,A -85,B 0,C 180,E1 -15818.915,E2 -15818.915} C_VEL
LIN {X 0,Y 312.623,Z 278.354,A -85,B 0,C 180,E1 -15821.658,E2 -15821.658} C_VEL
LIN {X 0,Y 312.586,Z 278.357,A -85,B 0,C 180,E1 -15823.18,E2 -15823.18} C_VEL
LIN {X 0,Y 311.906,Z 278.447,A -85,B 0,C 180,E1 -15824.255,E2 -15824.255} C_VEL
LIN {X 0,Y 309.053,Z 278.797,A -85,B 0,C 180,E1 -15826.007,E2 -15826.007} C_VEL
LIN {X 0,Y 306.66,Z 279.098,A -85,B 0,C 180,E1 -15827.428,E2 -15827.428} C_VEL
LIN {X 0,Y 305.66,Z 279.222,A -85,B 0,C 180,E1 -15828.527,E2 -15828.527} C_VEL
LIN {X 0,Y 305.593,Z 279.227,A -85,B 0,C 180,E1 -15828.9,E2 -15828.9} C_VEL
LIN {X 0,Y 305.75,Z 279.212,A -85,B 0,C 180,E1 -15832.075,E2 -15832.075} C_VEL
LIN {X 0,Y 305.665,Z 279.222,A -85,B 0,C 180,E1 -15834.726,E2 -15834.726} C_VEL
LIN {X 0,Y 305.948,Z 279.183,A -85,B 0,C 180,E1 -15838.686,E2 -15838.686} C_VEL
LIN {X 0,Y 305.946,Z 279.184,A -85,B 0,C 180,E1 -15841.319,E2 -15841.319} C_VEL
LIN {X 0,Y 305.843,Z 279.195,A -85,B 0,C 180,E1 -15846.6,E2 -15846.6} C_VEL
LIN {X 0,Y 305.727,Z 279.214,A -85,B 0,C 180,E1 -15849.262,E2 -15849.262} C_VEL
LIN {X 0,Y 305.582,Z 279.234,A -85,B 0,C 180,E1 -15853.298,E2 -15853.298} C_VEL
LIN {X 0,Y 305.586,Z 279.233,A -85,B 0,C 180,E1 -15856.023,E2 -15856.023} C_VEL
LIN {X 0,Y 305.568,Z 279.236,A -85,B 0,C 180,E1 -15859.447,E2 -15859.447} C_VEL
LIN {X 0,Y 305.48,Z 279.249,A -85,B 0,C 180,E1 -15863.042,E2 -15863.042} C_VEL
LIN {X 0,Y 305.466,Z 279.253,A -85,B 0,C 180,E1 -15866.201,E2 -15866.201} C_VEL
LIN {X 0,Y 305.444,Z 279.256,A -85,B 0,C 180,E1 -15869.037,E2 -15869.037} C_VEL
LIN {X 0,Y 305.431,Z 279.258,A -85,B 0,C 180,E1 -15871.956,E2 -15871.956} C_VEL
LIN {X 0,Y 305.458,Z 279.254,A -85,B 0,C 180,E1 -15875.116,E2 -15875.116} C_VEL
LIN {X 0,Y 305.478,Z 279.249,A -85,B 0,C 180,E1 -15878.539,E2 -15878.539} C_VEL
LIN {X 0,Y 305.484,Z 279.248,A -85,B 0,C 180,E1 -15882.595,E2 -15882.595} C_VEL
LIN {X 0,Y 305.457,Z 279.308,A -85,B 0,C 180,E1 -15884.082,E2 -15884.082} C_VEL
LIN {X 0,Y 306.304,Z 283.973,A -85,B 0,C 180,E1 -15888.29,E2 -15888.29} C_VEL
LIN {X 0,Y 307.054,Z 288.286,A -85,B 0,C 180,E1 -15891.833,E2 -15891.833} C_VEL
LIN {X 0,Y 307.552,Z 291.576,A -85,B 0,C 180,E1 -15894.361,E2 -15894.361} C_VEL
LIN {X 0,Y 307.677,Z 294.846,A -85,B 0,C 180,E1 -15896.758,E2 -15896.758} C_VEL
LIN {X 0,Y 306.744,Z 300.461,A -85,B 0,C 180,E1 -15900.536,E2 -15900.536} C_VEL
LIN {X 0,Y 305.663,Z 307.076,A -85,B 0,C 180,E1 -15904.828,E2 -15904.828} C_VEL
LIN {X 0,Y 304.769,Z 314.197,A -85,B 0,C 180,E1 -15909.28,E2 -15909.28} C_VEL
LIN {X 0,Y 307.568,Z 327.076,A -85,B 0,C 180,E1 -15910.22,E2 -15910.22} C_VEL
LIN {X 0,Y 309.052,Z 336.989,A -85,B 0,C 180,E1 -15911.133,E2 -15911.133} C_VEL
LIN {X 0,Y 309.719,Z 344.685,A -85,B 0,C 180,E1 -15911.964,E2 -15911.964} C_VEL
LIN {X 0,Y 309.914,Z 353.081,A -85,B 0,C 180,E1 -15913.026,E2 -15913.026} C_VEL
LIN {X 0,Y 309.269,Z 359.893,A -85,B 0,C 180,E1 -15914.008,E2 -15914.008} C_VEL
LIN {X 0,Y 308.091,Z 366.57,A -85,B 0,C 180,E1 -15915.132,E2 -15915.132} C_VEL
LIN {X 0,Y 306.967,Z 372.92,A -85,B 0,C 180,E1 -15916.43,E2 -15916.43} C_VEL
LIN {X 0,Y 306.063,Z 378.215,A -85,B 0,C 180,E1 -15917.739,E2 -15917.739} C_VEL
LIN {X 0,Y 305.105,Z 383.608,A -85,B 0,C 180,E1 -15919.383,E2 -15919.383} C_VEL
LIN {X 0,Y 304.544,Z 387.121,A -85,B 0,C 180,E1 -15920.706,E2 -15920.706} C_VEL
LIN {X 0,Y 303.977,Z 391.183,A -85,B 0,C 180,E1 -15922.696,E2 -15922.696} C_VEL
LIN {X 0,Y 303.695,Z 394.007,A -85,B 0,C 180,E1 -15924.691,E2 -15924.691} C_VEL
LIN {X 0,Y 303.692,Z 395.185,A -85,B 0,C 180,E1 -15926.021,E2 -15926.021} C_VEL
LIN {X 0,Y 303.667,Z 395.895,A -85,B 0,C 180,E1 -15927.349,E2 -15927.349} C_VEL
LIN {X 0,Y 303.686,Z 396.149,A -85,B 0,C 180,E1 -15928.676,E2 -15928.676} C_VEL
LIN {X 0,Y 303.767,Z 395.854,A -85,B 0,C 180,E1 -15930.002,E2 -15930.002} C_VEL
LIN {X 0,Y 303.73,Z 394.993,A -85,B 0,C 180,E1 -15931.328,E2 -15931.328} C_VEL
LIN {X 0,Y 303.707,Z 393.649,A -85,B 0,C 180,E1 -15932.654,E2 -15932.654} C_VEL
LIN {X 0,Y 303.775,Z 390.639,A -85,B 0,C 180,E1 -15934.646,E2 -15934.646} C_VEL
LIN {X 0,Y 303.863,Z 386.317,A -85,B 0,C 180,E1 -15936.642,E2 -15936.642} C_VEL
LIN {X 0,Y 304.248,Z 380.307,A -85,B 0,C 180,E1 -15938.637,E2 -15938.637} C_VEL
LIN {X 0,Y 304.542,Z 375.309,A -85,B 0,C 180,E1 -15939.969,E2 -15939.969} C_VEL
LIN {X 0,Y 305.109,Z 369.295,A -85,B 0,C 180,E1 -15941.293,E2 -15941.293} C_VEL
LIN {X 0,Y 305.768,Z 361.962,A -85,B 0,C 180,E1 -15942.614,E2 -15942.614} C_VEL
LIN {X 0,Y 306.451,Z 354.114,A -85,B 0,C 180,E1 -15943.766,E2 -15943.766} C_VEL
LIN {X 0,Y 306.665,Z 348.82,A -85,B 0,C 180,E1 -15944.433,E2 -15944.433} C_VEL
LIN {X 0,Y 306.174,Z 339.668,A -85,B 0,C 180,E1 -15945.399,E2 -15945.399} C_VEL
LIN {X 0,Y 305.614,Z 331.279,A -85,B 0,C 180,E1 -15946.106,E2 -15946.106} C_VEL
LIN {X 0,Y 304.779,Z 321.611,A -85,B 0,C 180,E1 -15946.733,E2 -15946.733} C_VEL
LIN {X 0,Y 304.063,Z 314.898,A -85,B 0,C 180,E1 -15947.098,E2 -15947.098} C_VEL
LIN {X 0,Y 304.608,Z 307.198,A -85,B 0,C 180,E1 -15951.665,E2 -15951.665} C_VEL
LIN {X 0,Y 305.335,Z 299.755,A -85,B 0,C 180,E1 -15956.143,E2 -15956.143} C_VEL
LIN {X 0,Y 306.219,Z 292.953,A -85,B 0,C 180,E1 -15960.328,E2 -15960.328} C_VEL
LIN {X 0,Y 306.828,Z 289.35,A -85,B 0,C 180,E1 -15962.599,E2 -15962.599} C_VEL
LIN {X 0,Y 306.709,Z 285.76,A -85,B 0,C 180,E1 -15964.951,E2 -15964.951} C_VEL
LIN {X 0,Y 305.746,Z 280.525,A -85,B 0,C 180,E1 -15968.596,E2 -15968.596} C_VEL
LIN {X 0,Y 305.516,Z 279.243,A -85,B 0,C 180,E1 -15969.6,E2 -15969.6} C_VEL
LIN {X 0,Y 305.436,Z 279.251,A -85,B 0,C 180,E1 -15973.655,E2 -15973.655} C_VEL
LIN {X 0,Y 305.465,Z 279.246,A -85,B 0,C 180,E1 -15977.414,E2 -15977.414} C_VEL
LIN {X 0,Y 305.486,Z 279.246,A -85,B 0,C 180,E1 -15981.597,E2 -15981.597} C_VEL
LIN {X 0,Y 305.473,Z 279.244,A -85,B 0,C 180,E1 -15984.886,E2 -15984.886} C_VEL
LIN {X 0,Y 305.462,Z 279.244,A -85,B 0,C 180,E1 -15988.354,E2 -15988.354} C_VEL
LIN {X 0,Y 305.531,Z 279.238,A -85,B 0,C 180,E1 -15991.113,E2 -15991.113} C_VEL
LIN {X 0,Y 305.582,Z 279.23,A -85,B 0,C 180,E1 -15994.087,E2 -15994.087} C_VEL
LIN {X 0,Y 305.484,Z 279.241,A -85,B 0,C 180,E1 -15998.4,E2 -15998.4} C_VEL
LIN {X 0,Y 305.527,Z 279.242,A -85,B 0,C 180,E1 -16001.212,E2 -16001.212} C_VEL
LIN {X 0,Y 305.635,Z 279.226,A -85,B 0,C 180,E1 -16005.346,E2 -16005.346} C_VEL
LIN {X 0,Y 305.633,Z 279.225,A -85,B 0,C 180,E1 -16009.397,E2 -16009.397} C_VEL
LIN {X 0,Y 305.78,Z 279.206,A -85,B 0,C 180,E1 -16012.071,E2 -16012.071} C_VEL
LIN {X 0,Y 305.69,Z 279.222,A -85,B 0,C 180,E1 -16014.721,E2 -16014.721} C_VEL
LIN {X 0,Y 305.962,Z 279.186,A -85,B 0,C 180,E1 -16018.681,E2 -16018.681} C_VEL
LIN {X 0,Y 305.964,Z 279.182,A -85,B 0,C 180,E1 -16021.314,E2 -16021.314} C_VEL
LIN {X 0,Y 305.858,Z 279.199,A -85,B 0,C 180,E1 -16026.595,E2 -16026.595} C_VEL
LIN {X 0,Y 305.741,Z 279.209,A -85,B 0,C 180,E1 -16029.257,E2 -16029.257} C_VEL
LIN {X 0,Y 305.592,Z 279.228,A -85,B 0,C 180,E1 -16033.293,E2 -16033.293} C_VEL
LIN {X 0,Y 305.596,Z 279.233,A -85,B 0,C 180,E1 -16036.017,E2 -16036.017} C_VEL
LIN {X 0,Y 305.578,Z 279.231,A -85,B 0,C 180,E1 -16039.442,E2 -16039.442} C_VEL
LIN {X 0,Y 305.491,Z 279.241,A -85,B 0,C 180,E1 -16043.038,E2 -16043.038} C_VEL
LIN {X 0,Y 305.531,Z 279.239,A -85,B 0,C 180,E1 -16046.218,E2 -16046.218} C_VEL
LIN {X 0,Y 305.486,Z 279.242,A -85,B 0,C 180,E1 -16049.044,E2 -16049.044} C_VEL
LIN {X 0,Y 305.44,Z 279.251,A -85,B 0,C 180,E1 -16051.949,E2 -16051.949} C_VEL
LIN {X 0,Y 305.459,Z 279.247,A -85,B 0,C 180,E1 -16055.11,E2 -16055.11} C_VEL
LIN {X 0,Y 305.489,Z 279.242,A -85,B 0,C 180,E1 -16058.536,E2 -16058.536} C_VEL
LIN {X 0,Y 305.516,Z 279.239,A -85,B 0,C 180,E1 -16062.596,E2 -16062.596} C_VEL
LIN {X 0,Y 305.526,Z 279.237,A -85,B 0,C 180,E1 -16066.361,E2 -16066.361} C_VEL
LIN {X 0,Y 305.476,Z 279.243,A -85,B 0,C 180,E1 -16069.893,E2 -16069.893} C_VEL
LIN {X 0,Y 305.49,Z 279.242,A -85,B 0,C 180,E1 -16073.624,E2 -16073.624} C_VEL
LIN {X 0,Y 305.454,Z 279.248,A -85,B 0,C 180,E1 -16076.48,E2 -16076.48} C_VEL
LIN {X 0,Y 305.484,Z 279.246,A -85,B 0,C 180,E1 -16080.947,E2 -16080.947} C_VEL
LIN {X 0,Y 305.56,Z 279.234,A -85,B 0,C 180,E1 -16084.085,E2 -16084.085} C_VEL
LIN {X 0,Y 305.476,Z 279.247,A -85,B 0,C 180,E1 -16088.399,E2 -16088.399} C_VEL
LIN {X 0,Y 305.419,Z 279.25,A -85,B 0,C 180,E1 -16091.205,E2 -16091.205} C_VEL
LIN {X 0,Y 305.026,Z 279.299,A -85,B 0,C 180,E1 -16095.386,E2 -16095.386} C_VEL
LIN {X 0,Y 304.827,Z 279.328,A -85,B 0,C 180,E1 -16096.668,E2 -16096.668} C_VEL
LIN {X 0,Y 304.631,Z 281.531,A -85,B 0,C 180,E1 -16099.363,E2 -16099.363} C_VEL
LIN {X 0,Y 304.634,Z 285.493,A -85,B 0,C 180,E1 -16103.374,E2 -16103.374} C_VEL
LIN {X 0,Y 304.421,Z 289.201,A -85,B 0,C 180,E1 -16107.021,E2 -16107.021} C_VEL
LIN {X 0,Y 304.571,Z 290.426,A -85,B 0,C 180,E1 -16107.146,E2 -16107.146} C_VEL
LIN {X 0,Y 306.282,Z 300.464,A -85,B 0,C 180,E1 -16107.779,E2 -16107.779} C_VEL
LIN {X 0,Y 307.489,Z 309.554,A -85,B 0,C 180,E1 -16108.525,E2 -16108.525} C_VEL
LIN {X 0,Y 308.052,Z 314.731,A -85,B 0,C 180,E1 -16109.018,E2 -16109.018} C_VEL
LIN {X 0,Y 307.217,Z 324.813,A -85,B 0,C 180,E1 -16110.162,E2 -16110.162} C_VEL
LIN {X 0,Y 306.54,Z 332.839,A -85,B 0,C 180,E1 -16111.312,E2 -16111.312} C_VEL
LIN {X 0,Y 306.012,Z 338.611,A -85,B 0,C 180,E1 -16112.302,E2 -16112.302} C_VEL
LIN {X 0,Y 305.463,Z 345.034,A -85,B 0,C 180,E1 -16113.626,E2 -16113.626} C_VEL
LIN {X 0,Y 304.849,Z 351.568,A -85,B 0,C 180,E1 -16115.289,E2 -16115.289} C_VEL
LIN {X 0,Y 304.533,Z 355.807,A -85,B 0,C 180,E1 -16116.624,E2 -16116.624} C_VEL
LIN {X 0,Y 304.219,Z 359.328,A -85,B 0,C 180,E1 -16117.966,E2 -16117.966} C_VEL
LIN {X 0,Y 303.833,Z 363.385,A -85,B 0,C 180,E1 -16119.989,E2 -16119.989} C_VEL
LIN {X 0,Y 303.671,Z 366.165,A -85,B 0,C 180,E1 -16122.02,E2 -16122.02} C_VEL
LIN {X 0,Y 303.653,Z 367.409,A -85,B 0,C 180,E1 -16123.585,E2 -16123.585} C_VEL
LIN {X 0,Y 303.675,Z 367.857,A -85,B 0,C 180,E1 -16124.746,E2 -16124.746} C_VEL
LIN {X 0,Y 303.737,Z 367.967,A -85,B 0,C 180,E1 -16126.119,E2 -16126.119} C_VEL
LIN {X 0,Y 303.954,Z 367.577,A -85,B 0,C 180,E1 -16127.491,E2 -16127.491} C_VEL
LIN {X 0,Y 304.25,Z 366.609,A -85,B 0,C 180,E1 -16128.866,E2 -16128.866} C_VEL
LIN {X 0,Y 304.843,Z 364.084,A -85,B 0,C 180,E1 -16130.935,E2 -16130.935} C_VEL
LIN {X 0,Y 305.371,Z 361.694,A -85,B 0,C 180,E1 -16132.316,E2 -16132.316} C_VEL
LIN {X 0,Y 306.354,Z 356.726,A -85,B 0,C 180,E1 -16134.387,E2 -16134.387} C_VEL
LIN {X 0,Y 307.205,Z 352.517,A -85,B 0,C 180,E1 -16135.762,E2 -16135.762} C_VEL
LIN {X 0,Y 308.192,Z 347.051,A -85,B 0,C 180,E1 -16137.215,E2 -16137.215} C_VEL
LIN {X 0,Y 309.22,Z 341.125,A -85,B 0,C 180,E1 -16138.506,E2 -16138.506} C_VEL
LIN {X 0,Y 310.32,Z 334.509,A -85,B 0,C 180,E1 -16139.695,E2 -16139.695} C_VEL
LIN {X 0,Y 311.421,Z 327.763,A -85,B 0,C 180,E1 -16140.695,E2 -16140.695} C_VEL
LIN {X 0,Y 312.234,Z 321.415,A -85,B 0,C 180,E1 -16141.498,E2 -16141.498} C_VEL
LIN {X 0,Y 310.784,Z 312.353,A -85,B 0,C 180,E1 -16142.617,E2 -16142.617} C_VEL
LIN {X 0,Y 308.743,Z 303.752,A -85,B 0,C 180,E1 -16143.538,E2 -16143.538} C_VEL
LIN {X 0,Y 305.984,Z 294.777,A -85,B 0,C 180,E1 -16144.37,E2 -16144.37} C_VEL
LIN {X 0,Y 304.563,Z 290.024,A -85,B 0,C 180,E1 -16144.781,E2 -16144.781} C_VEL
LIN {X 0,Y 304.862,Z 286.642,A -85,B 0,C 180,E1 -16148.491,E2 -16148.491} C_VEL
LIN {X 0,Y 305.215,Z 283.106,A -85,B 0,C 180,E1 -16152.541,E2 -16152.541} C_VEL
LIN {X 0,Y 305.317,Z 279.939,A -85,B 0,C 180,E1 -16156.33,E2 -16156.33} C_VEL
LIN {X 0,Y 305.281,Z 279.27,A -85,B 0,C 180,E1 -16157.447,E2 -16157.447} C_VEL
LIN {X 0,Y 305.403,Z 279.257,A -85,B 0,C 180,E1 -16159.888,E2 -16159.888} C_VEL
LIN {X 0,Y 305.481,Z 279.249,A -85,B 0,C 180,E1 -16163.628,E2 -16163.628} C_VEL
LIN {X 0,Y 305.446,Z 279.251,A -85,B 0,C 180,E1 -16166.485,E2 -16166.485} C_VEL
LIN {X 0,Y 305.44,Z 279.251,A -85,B 0,C 180,E1 -16169.592,E2 -16169.592} C_VEL
LIN {X 0,Y 305.501,Z 279.244,A -85,B 0,C 180,E1 -16172.61,E2 -16172.61} C_VEL
LIN {X 0,Y 305.489,Z 279.244,A -85,B 0,C 180,E1 -16175.54,E2 -16175.54} C_VEL
LIN {X 0,Y 305.497,Z 279.242,A -85,B 0,C 180,E1 -16179.816,E2 -16179.816} C_VEL
LIN {X 0,Y 305.546,Z 279.232,A -85,B 0,C 180,E1 -16183.18,E2 -16183.18} C_VEL
LIN {X 0,Y 305.635,Z 279.222,A -85,B 0,C 180,E1 -16185.351,E2 -16185.351} C_VEL
LIN {X 0,Y 305.593,Z 279.227,A -85,B 0,C 180,E1 -16188.9,E2 -16188.9} C_VEL
LIN {X 0,Y 304.981,Z 279.304,A -85,B 0,C 180,E1 -16190,E2 -16190} C_VEL
LIN {X 0,Y 302.206,Z 279.654,A -85,B 0,C 180,E1 -16191.794,E2 -16191.794} C_VEL
LIN {X 0,Y 299.801,Z 279.953,A -85,B 0,C 180,E1 -16193.249,E2 -16193.249} C_VEL
LIN {X 0,Y 298.727,Z 280.085,A -85,B 0,C 180,E1 -16194.374,E2 -16194.374} C_VEL
LIN {X 0,Y 298.619,Z 280.097,A -85,B 0,C 180,E1 -16194.756,E2 -16194.756} C_VEL
LIN {X 0,Y 298.914,Z 280.059,A -85,B 0,C 180,E1 -16198.655,E2 -16198.655} C_VEL
LIN {X 0,Y 298.912,Z 280.06,A -85,B 0,C 180,E1 -16201.35,E2 -16201.35} C_VEL
LIN {X 0,Y 298.788,Z 280.074,A -85,B 0,C 180,E1 -16206.756,E2 -16206.756} C_VEL
LIN {X 0,Y 298.672,Z 280.093,A -85,B 0,C 180,E1 -16209.483,E2 -16209.483} C_VEL
